Fanuc TP program (LS listing): surfaceorigin.ls

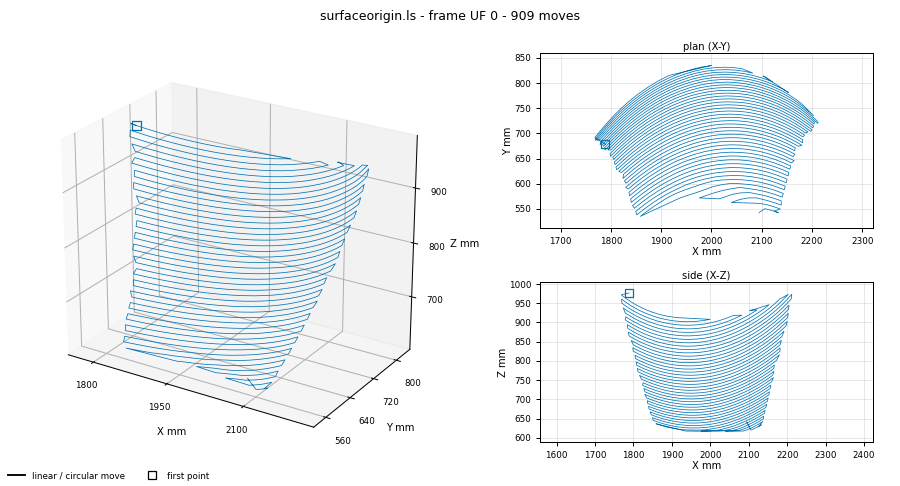
[picture p0: tool path of surfaceorigin.ls in frame UF 0, 909 of 909 moves have a stored position in this frame; points joined in program order, loops and branches not executed]
/PROG surfaceorigin
/ATTR
OWNER			= MNEDITOR;
COMMENT			= "";
PROG_SIZE		= 4757;
FILE_NAME		= surface;
VERSION			= 0;
LINE_COUNT		= 909;
MEMORY_SIZE		= 5089;
PROTECT			= READ_WRITE;
TCD:  STACK_SIZE		= 0,
      TASK_PRIORITY		= 50,
      TIME_SLICE		= 0,
      BUSY_LAMP_OFF		= 0,
      ABORT_REQUEST		= 0,
      PAUSE_REQUEST		= 0;
DEFAULT_GROUP	= 1,*,*,*,*;
CONTROL_CODE	= 00000000 00000000;
/MN
	1:  UFRAME_NUM=0 ;
	2:  UTOOL_NUM=1 ;
	3:	;
	4:	;
	5:J P[1] 100% CNT60 	;
	6:L P[2] 200mm/sec CNT60 	;
	7:L P[3] 200mm/sec CNT60 	;
	8:L P[4] 200mm/sec CNT60 	;
	9:L P[5] 200mm/sec CNT60 	;
	10:L P[6] 200mm/sec CNT60 	;
	11:L P[7] 200mm/sec CNT60 	;
	12:L P[8] 200mm/sec CNT60 	;
	13:L P[9] 200mm/sec CNT60 	;
	14:L P[10] 200mm/sec CNT60 	;
	15:L P[11] 200mm/sec CNT60 	;
	16:L P[12] 200mm/sec CNT60 	;
	17:L P[13] 200mm/sec CNT60 	;
	18:L P[14] 200mm/sec CNT60 	;
	19:L P[15] 200mm/sec CNT60 	;
	20:L P[16] 200mm/sec CNT60 	;
	21:L P[17] 200mm/sec CNT60 	;
	22:L P[18] 200mm/sec CNT60 	;
	23:L P[19] 200mm/sec CNT60 	;
	24:L P[20] 200mm/sec CNT60 	;
	25:L P[21] 200mm/sec CNT60 	;
	26:L P[22] 200mm/sec CNT60 	;
	27:L P[23] 200mm/sec CNT60 	;
	28:L P[24] 200mm/sec CNT60 	;
	29:L P[25] 200mm/sec CNT60 	;
	30:L P[26] 200mm/sec CNT60 	;
	31:L P[27] 200mm/sec CNT60 	;
	32:L P[28] 200mm/sec CNT60 	;
	33:L P[29] 200mm/sec CNT60 	;
	34:L P[30] 200mm/sec CNT60 	;
	35:L P[31] 200mm/sec CNT60 	;
	36:L P[32] 200mm/sec CNT60 	;
	37:L P[33] 200mm/sec CNT60 	;
	38:L P[34] 200mm/sec CNT60 	;
	39:L P[35] 200mm/sec CNT60 	;
	40:L P[36] 200mm/sec CNT60 	;
	41:L P[37] 200mm/sec CNT60 	;
	42:L P[38] 200mm/sec CNT60 	;
	43:L P[39] 200mm/sec CNT60 	;
	44:L P[40] 200mm/sec CNT60 	;
	45:L P[41] 200mm/sec CNT60 	;
	46:L P[42] 200mm/sec CNT60 	;
	47:L P[43] 200mm/sec CNT60 	;
	48:L P[44] 200mm/sec CNT60 	;
	49:L P[45] 200mm/sec CNT60 	;
	50:L P[46] 200mm/sec CNT60 	;
	51:L P[47] 200mm/sec CNT60 	;
	52:L P[48] 200mm/sec CNT60 	;
	53:L P[49] 200mm/sec CNT60 	;
	54:L P[50] 200mm/sec CNT60 	;
	55:L P[51] 200mm/sec CNT60 	;
	56:L P[52] 200mm/sec CNT60 	;
	57:L P[53] 200mm/sec CNT60 	;
	58:L P[54] 200mm/sec CNT60 	;
	59:L P[55] 200mm/sec CNT60 	;
	60:L P[56] 200mm/sec CNT60 	;
	61:L P[57] 200mm/sec CNT60 	;
	62:L P[58] 200mm/sec CNT60 	;
	63:L P[59] 200mm/sec CNT60 	;
	64:L P[60] 200mm/sec CNT60 	;
	65:L P[61] 200mm/sec CNT60 	;
	66:L P[62] 200mm/sec CNT60 	;
	67:L P[63] 200mm/sec CNT60 	;
	68:L P[64] 200mm/sec CNT60 	;
	69:L P[65] 200mm/sec CNT60 	;
	70:L P[66] 200mm/sec CNT60 	;
	71:L P[67] 200mm/sec CNT60 	;
	72:L P[68] 200mm/sec CNT60 	;
	73:L P[69] 200mm/sec CNT60 	;
	74:L P[70] 200mm/sec CNT60 	;
	75:L P[71] 200mm/sec CNT60 	;
	76:L P[72] 200mm/sec CNT60 	;
	77:L P[73] 200mm/sec CNT60 	;
	78:L P[74] 200mm/sec CNT60 	;
	79:L P[75] 200mm/sec CNT60 	;
	80:L P[76] 200mm/sec CNT60 	;
	81:L P[77] 200mm/sec CNT60 	;
	82:L P[78] 200mm/sec CNT60 	;
	83:L P[79] 200mm/sec CNT60 	;
	84:L P[80] 200mm/sec CNT60 	;
	85:L P[81] 200mm/sec CNT60 	;
	86:L P[82] 200mm/sec CNT60 	;
	87:L P[83] 200mm/sec CNT60 	;
	88:L P[84] 200mm/sec CNT60 	;
	89:L P[85] 200mm/sec CNT60 	;
	90:L P[86] 200mm/sec CNT60 	;
	91:L P[87] 200mm/sec CNT60 	;
	92:L P[88] 200mm/sec CNT60 	;
	93:L P[89] 200mm/sec CNT60 	;
	94:L P[90] 200mm/sec CNT60 	;
	95:L P[91] 200mm/sec CNT60 	;
	96:L P[92] 200mm/sec CNT60 	;
	97:L P[93] 200mm/sec CNT60 	;
	98:L P[94] 200mm/sec CNT60 	;
	99:L P[95] 200mm/sec CNT60 	;
	100:L P[96] 200mm/sec CNT60 	;
	101:L P[97] 200mm/sec CNT60 	;
	102:L P[98] 200mm/sec CNT60 	;
	103:L P[99] 200mm/sec CNT60 	;
	104:L P[100] 200mm/sec CNT60 	;
	105:L P[101] 200mm/sec CNT60 	;
	106:L P[102] 200mm/sec CNT60 	;
	107:L P[103] 200mm/sec CNT60 	;
	108:L P[104] 200mm/sec CNT60 	;
	109:L P[105] 200mm/sec CNT60 	;
	110:L P[106] 200mm/sec CNT60 	;
	111:L P[107] 200mm/sec CNT60 	;
	112:L P[108] 200mm/sec CNT60 	;
	113:L P[109] 200mm/sec CNT60 	;
	114:L P[110] 200mm/sec CNT60 	;
	115:L P[111] 200mm/sec CNT60 	;
	116:L P[112] 200mm/sec CNT60 	;
	117:L P[113] 200mm/sec CNT60 	;
	118:L P[114] 200mm/sec CNT60 	;
	119:L P[115] 200mm/sec CNT60 	;
	120:L P[116] 200mm/sec CNT60 	;
	121:L P[117] 200mm/sec CNT60 	;
	122:L P[118] 200mm/sec CNT60 	;
	123:L P[119] 200mm/sec CNT60 	;
	124:L P[120] 200mm/sec CNT60 	;
	125:L P[121] 200mm/sec CNT60 	;
	126:L P[122] 200mm/sec CNT60 	;
	127:L P[123] 200mm/sec CNT60 	;
	128:L P[124] 200mm/sec CNT60 	;
	129:L P[125] 200mm/sec CNT60 	;
	130:L P[126] 200mm/sec CNT60 	;
	131:L P[127] 200mm/sec CNT60 	;
	132:L P[128] 200mm/sec CNT60 	;
	133:L P[129] 200mm/sec CNT60 	;
	134:L P[130] 200mm/sec CNT60 	;
	135:L P[131] 200mm/sec CNT60 	;
	136:L P[132] 200mm/sec CNT60 	;
	137:L P[133] 200mm/sec CNT60 	;
	138:L P[134] 200mm/sec CNT60 	;
	139:L P[135] 200mm/sec CNT60 	;
	140:L P[136] 200mm/sec CNT60 	;
	141:L P[137] 200mm/sec CNT60 	;
	142:L P[138] 200mm/sec CNT60 	;
	143:L P[139] 200mm/sec CNT60 	;
	144:L P[140] 200mm/sec CNT60 	;
	145:L P[141] 200mm/sec CNT60 	;
	146:L P[142] 200mm/sec CNT60 	;
	147:L P[143] 200mm/sec CNT60 	;
	148:L P[144] 200mm/sec CNT60 	;
	149:L P[145] 200mm/sec CNT60 	;
	150:L P[146] 200mm/sec CNT60 	;
	151:L P[147] 200mm/sec CNT60 	;
	152:L P[148] 200mm/sec CNT60 	;
	153:L P[149] 200mm/sec CNT60 	;
	154:L P[150] 200mm/sec CNT60 	;
	155:L P[151] 200mm/sec CNT60 	;
	156:L P[152] 200mm/sec CNT60 	;
	157:L P[153] 200mm/sec CNT60 	;
	158:L P[154] 200mm/sec CNT60 	;
	159:L P[155] 200mm/sec CNT60 	;
	160:L P[156] 200mm/sec CNT60 	;
	161:L P[157] 200mm/sec CNT60 	;
	162:L P[158] 200mm/sec CNT60 	;
	163:L P[159] 200mm/sec CNT60 	;
	164:L P[160] 200mm/sec CNT60 	;
	165:L P[161] 200mm/sec CNT60 	;
	166:L P[162] 200mm/sec CNT60 	;
	167:L P[163] 200mm/sec CNT60 	;
	168:L P[164] 200mm/sec CNT60 	;
	169:L P[165] 200mm/sec CNT60 	;
	170:L P[166] 200mm/sec CNT60 	;
	171:L P[167] 200mm/sec CNT60 	;
	172:L P[168] 200mm/sec CNT60 	;
	173:L P[169] 200mm/sec CNT60 	;
	174:L P[170] 200mm/sec CNT60 	;
	175:L P[171] 200mm/sec CNT60 	;
	176:L P[172] 200mm/sec CNT60 	;
	177:L P[173] 200mm/sec CNT60 	;
	178:L P[174] 200mm/sec CNT60 	;
	179:L P[175] 200mm/sec CNT60 	;
	180:L P[176] 200mm/sec CNT60 	;
	181:L P[177] 200mm/sec CNT60 	;
	182:L P[178] 200mm/sec CNT60 	;
	183:L P[179] 200mm/sec CNT60 	;
	184:L P[180] 200mm/sec CNT60 	;
	185:L P[181] 200mm/sec CNT60 	;
	186:L P[182] 200mm/sec CNT60 	;
	187:L P[183] 200mm/sec CNT60 	;
	188:L P[184] 200mm/sec CNT60 	;
	189:L P[185] 200mm/sec CNT60 	;
	190:L P[186] 200mm/sec CNT60 	;
	191:L P[187] 200mm/sec CNT60 	;
	192:L P[188] 200mm/sec CNT60 	;
	193:L P[189] 200mm/sec CNT60 	;
	194:L P[190] 200mm/sec CNT60 	;
	195:L P[191] 200mm/sec CNT60 	;
	196:L P[192] 200mm/sec CNT60 	;
	197:L P[193] 200mm/sec CNT60 	;
	198:L P[194] 200mm/sec CNT60 	;
	199:L P[195] 200mm/sec CNT60 	;
	200:L P[196] 200mm/sec CNT60 	;
	201:L P[197] 200mm/sec CNT60 	;
	202:L P[198] 200mm/sec CNT60 	;
	203:L P[199] 200mm/sec CNT60 	;
	204:L P[200] 200mm/sec CNT60 	;
	205:L P[201] 200mm/sec CNT60 	;
	206:L P[202] 200mm/sec CNT60 	;
	207:L P[203] 200mm/sec CNT60 	;
	208:L P[204] 200mm/sec CNT60 	;
	209:L P[205] 200mm/sec CNT60 	;
	210:L P[206] 200mm/sec CNT60 	;
	211:L P[207] 200mm/sec CNT60 	;
	212:L P[208] 200mm/sec CNT60 	;
	213:L P[209] 200mm/sec CNT60 	;
	214:L P[210] 200mm/sec CNT60 	;
	215:L P[211] 200mm/sec CNT60 	;
	216:L P[212] 200mm/sec CNT60 	;
	217:L P[213] 200mm/sec CNT60 	;
	218:L P[214] 200mm/sec CNT60 	;
	219:L P[215] 200mm/sec CNT60 	;
	220:L P[216] 200mm/sec CNT60 	;
	221:L P[217] 200mm/sec CNT60 	;
	222:L P[218] 200mm/sec CNT60 	;
	223:L P[219] 200mm/sec CNT60 	;
	224:L P[220] 200mm/sec CNT60 	;
	225:L P[221] 200mm/sec CNT60 	;
	226:L P[222] 200mm/sec CNT60 	;
	227:L P[223] 200mm/sec CNT60 	;
	228:L P[224] 200mm/sec CNT60 	;
	229:L P[225] 200mm/sec CNT60 	;
	230:L P[226] 200mm/sec CNT60 	;
	231:L P[227] 200mm/sec CNT60 	;
	232:L P[228] 200mm/sec CNT60 	;
	233:L P[229] 200mm/sec CNT60 	;
	234:L P[230] 200mm/sec CNT60 	;
	235:L P[231] 200mm/sec CNT60 	;
	236:L P[232] 200mm/sec CNT60 	;
	237:L P[233] 200mm/sec CNT60 	;
	238:L P[234] 200mm/sec CNT60 	;
	239:L P[235] 200mm/sec CNT60 	;
	240:L P[236] 200mm/sec CNT60 	;
	241:L P[237] 200mm/sec CNT60 	;
	242:L P[238] 200mm/sec CNT60 	;
	243:L P[239] 200mm/sec CNT60 	;
	244:L P[240] 200mm/sec CNT60 	;
	245:L P[241] 200mm/sec CNT60 	;
	246:L P[242] 200mm/sec CNT60 	;
	247:L P[243] 200mm/sec CNT60 	;
	248:L P[244] 200mm/sec CNT60 	;
	249:L P[245] 200mm/sec CNT60 	;
	250:L P[246] 200mm/sec CNT60 	;
	251:L P[247] 200mm/sec CNT60 	;
	252:L P[248] 200mm/sec CNT60 	;
	253:L P[249] 200mm/sec CNT60 	;
	254:L P[250] 200mm/sec CNT60 	;
	255:L P[251] 200mm/sec CNT60 	;
	256:L P[252] 200mm/sec CNT60 	;
	257:L P[253] 200mm/sec CNT60 	;
	258:L P[254] 200mm/sec CNT60 	;
	259:L P[255] 200mm/sec CNT60 	;
	260:L P[256] 200mm/sec CNT60 	;
	261:L P[257] 200mm/sec CNT60 	;
	262:L P[258] 200mm/sec CNT60 	;
	263:L P[259] 200mm/sec CNT60 	;
	264:L P[260] 200mm/sec CNT60 	;
	265:L P[261] 200mm/sec CNT60 	;
	266:L P[262] 200mm/sec CNT60 	;
	267:L P[263] 200mm/sec CNT60 	;
	268:L P[264] 200mm/sec CNT60 	;
	269:L P[265] 200mm/sec CNT60 	;
	270:L P[266] 200mm/sec CNT60 	;
	271:L P[267] 200mm/sec CNT60 	;
	272:L P[268] 200mm/sec CNT60 	;
	273:L P[269] 200mm/sec CNT60 	;
	274:L P[270] 200mm/sec CNT60 	;
	275:L P[271] 200mm/sec CNT60 	;
	276:L P[272] 200mm/sec CNT60 	;
	277:L P[273] 200mm/sec CNT60 	;
	278:L P[274] 200mm/sec CNT60 	;
	279:L P[275] 200mm/sec CNT60 	;
	280:L P[276] 200mm/sec CNT60 	;
	281:L P[277] 200mm/sec CNT60 	;
	282:L P[278] 200mm/sec CNT60 	;
	283:L P[279] 200mm/sec CNT60 	;
	284:L P[280] 200mm/sec CNT60 	;
	285:L P[281] 200mm/sec CNT60 	;
	286:L P[282] 200mm/sec CNT60 	;
	287:L P[283] 200mm/sec CNT60 	;
	288:L P[284] 200mm/sec CNT60 	;
	289:L P[285] 200mm/sec CNT60 	;
	290:L P[286] 200mm/sec CNT60 	;
	291:L P[287] 200mm/sec CNT60 	;
	292:L P[288] 200mm/sec CNT60 	;
	293:L P[289] 200mm/sec CNT60 	;
	294:L P[290] 200mm/sec CNT60 	;
	295:L P[291] 200mm/sec CNT60 	;
	296:L P[292] 200mm/sec CNT60 	;
	297:L P[293] 200mm/sec CNT60 	;
	298:L P[294] 200mm/sec CNT60 	;
	299:L P[295] 200mm/sec CNT60 	;
	300:L P[296] 200mm/sec CNT60 	;
	301:L P[297] 200mm/sec CNT60 	;
	302:L P[298] 200mm/sec CNT60 	;
	303:L P[299] 200mm/sec CNT60 	;
	304:L P[300] 200mm/sec CNT60 	;
	305:L P[301] 200mm/sec CNT60 	;
	306:L P[302] 200mm/sec CNT60 	;
	307:L P[303] 200mm/sec CNT60 	;
	308:L P[304] 200mm/sec CNT60 	;
	309:L P[305] 200mm/sec CNT60 	;
	310:L P[306] 200mm/sec CNT60 	;
	311:L P[307] 200mm/sec CNT60 	;
	312:L P[308] 200mm/sec CNT60 	;
	313:L P[309] 200mm/sec CNT60 	;
	314:L P[310] 200mm/sec CNT60 	;
	315:L P[311] 200mm/sec CNT60 	;
	316:L P[312] 200mm/sec CNT60 	;
	317:L P[313] 200mm/sec CNT60 	;
	318:L P[314] 200mm/sec CNT60 	;
	319:L P[315] 200mm/sec CNT60 	;
	320:L P[316] 200mm/sec CNT60 	;
	321:L P[317] 200mm/sec CNT60 	;
	322:L P[318] 200mm/sec CNT60 	;
	323:L P[319] 200mm/sec CNT60 	;
	324:L P[320] 200mm/sec CNT60 	;
	325:L P[321] 200mm/sec CNT60 	;
	326:L P[322] 200mm/sec CNT60 	;
	327:L P[323] 200mm/sec CNT60 	;
	328:L P[324] 200mm/sec CNT60 	;
	329:L P[325] 200mm/sec CNT60 	;
	330:L P[326] 200mm/sec CNT60 	;
	331:L P[327] 200mm/sec CNT60 	;
	332:L P[328] 200mm/sec CNT60 	;
	333:L P[329] 200mm/sec CNT60 	;
	334:L P[330] 200mm/sec CNT60 	;
	335:L P[331] 200mm/sec CNT60 	;
	336:L P[332] 200mm/sec CNT60 	;
	337:L P[333] 200mm/sec CNT60 	;
	338:L P[334] 200mm/sec CNT60 	;
	339:L P[335] 200mm/sec CNT60 	;
	340:L P[336] 200mm/sec CNT60 	;
	341:L P[337] 200mm/sec CNT60 	;
	342:L P[338] 200mm/sec CNT60 	;
	343:L P[339] 200mm/sec CNT60 	;
	344:L P[340] 200mm/sec CNT60 	;
	345:L P[341] 200mm/sec CNT60 	;
	346:L P[342] 200mm/sec CNT60 	;
	347:L P[343] 200mm/sec CNT60 	;
	348:L P[344] 200mm/sec CNT60 	;
	349:L P[345] 200mm/sec CNT60 	;
	350:L P[346] 200mm/sec CNT60 	;
	351:L P[347] 200mm/sec CNT60 	;
	352:L P[348] 200mm/sec CNT60 	;
	353:L P[349] 200mm/sec CNT60 	;
	354:L P[350] 200mm/sec CNT60 	;
	355:L P[351] 200mm/sec CNT60 	;
	356:L P[352] 200mm/sec CNT60 	;
	357:L P[353] 200mm/sec CNT60 	;
	358:L P[354] 200mm/sec CNT60 	;
	359:L P[355] 200mm/sec CNT60 	;
	360:L P[356] 200mm/sec CNT60 	;
	361:L P[357] 200mm/sec CNT60 	;
	362:L P[358] 200mm/sec CNT60 	;
	363:L P[359] 200mm/sec CNT60 	;
	364:L P[360] 200mm/sec CNT60 	;
	365:L P[361] 200mm/sec CNT60 	;
	366:L P[362] 200mm/sec CNT60 	;
	367:L P[363] 200mm/sec CNT60 	;
	368:L P[364] 200mm/sec CNT60 	;
	369:L P[365] 200mm/sec CNT60 	;
	370:L P[366] 200mm/sec CNT60 	;
	371:L P[367] 200mm/sec CNT60 	;
	372:L P[368] 200mm/sec CNT60 	;
	373:L P[369] 200mm/sec CNT60 	;
	374:L P[370] 200mm/sec CNT60 	;
	375:L P[371] 200mm/sec CNT60 	;
	376:L P[372] 200mm/sec CNT60 	;
	377:L P[373] 200mm/sec CNT60 	;
	378:L P[374] 200mm/sec CNT60 	;
	379:L P[375] 200mm/sec CNT60 	;
	380:L P[376] 200mm/sec CNT60 	;
	381:L P[377] 200mm/sec CNT60 	;
	382:L P[378] 200mm/sec CNT60 	;
	383:L P[379] 200mm/sec CNT60 	;
	384:L P[380] 200mm/sec CNT60 	;
	385:L P[381] 200mm/sec CNT60 	;
	386:L P[382] 200mm/sec CNT60 	;
	387:L P[383] 200mm/sec CNT60 	;
	388:L P[384] 200mm/sec CNT60 	;
	389:L P[385] 200mm/sec CNT60 	;
	390:L P[386] 200mm/sec CNT60 	;
	391:L P[387] 200mm/sec CNT60 	;
	392:L P[388] 200mm/sec CNT60 	;
	393:L P[389] 200mm/sec CNT60 	;
	394:L P[390] 200mm/sec CNT60 	;
	395:L P[391] 200mm/sec CNT60 	;
	396:L P[392] 200mm/sec CNT60 	;
	397:L P[393] 200mm/sec CNT60 	;
	398:L P[394] 200mm/sec CNT60 	;
	399:L P[395] 200mm/sec CNT60 	;
	400:L P[396] 200mm/sec CNT60 	;
	401:L P[397] 200mm/sec CNT60 	;
	402:L P[398] 200mm/sec CNT60 	;
	403:L P[399] 200mm/sec CNT60 	;
	404:L P[400] 200mm/sec CNT60 	;
	405:L P[401] 200mm/sec CNT60 	;
	406:L P[402] 200mm/sec CNT60 	;
	407:L P[403] 200mm/sec CNT60 	;
	408:L P[404] 200mm/sec CNT60 	;
	409:L P[405] 200mm/sec CNT60 	;
	410:L P[406] 200mm/sec CNT60 	;
	411:L P[407] 200mm/sec CNT60 	;
	412:L P[408] 200mm/sec CNT60 	;
	413:L P[409] 200mm/sec CNT60 	;
	414:L P[410] 200mm/sec CNT60 	;
	415:L P[411] 200mm/sec CNT60 	;
	416:L P[412] 200mm/sec CNT60 	;
	417:L P[413] 200mm/sec CNT60 	;
	418:L P[414] 200mm/sec CNT60 	;
	419:L P[415] 200mm/sec CNT60 	;
	420:L P[416] 200mm/sec CNT60 	;
	421:L P[417] 200mm/sec CNT60 	;
	422:L P[418] 200mm/sec CNT60 	;
	423:L P[419] 200mm/sec CNT60 	;
	424:L P[420] 200mm/sec CNT60 	;
	425:L P[421] 200mm/sec CNT60 	;
	426:L P[422] 200mm/sec CNT60 	;
	427:L P[423] 200mm/sec CNT60 	;
	428:L P[424] 200mm/sec CNT60 	;
	429:L P[425] 200mm/sec CNT60 	;
	430:L P[426] 200mm/sec CNT60 	;
	431:L P[427] 200mm/sec CNT60 	;
	432:L P[428] 200mm/sec CNT60 	;
	433:L P[429] 200mm/sec CNT60 	;
	434:L P[430] 200mm/sec CNT60 	;
	435:L P[431] 200mm/sec CNT60 	;
	436:L P[432] 200mm/sec CNT60 	;
	437:L P[433] 200mm/sec CNT60 	;
	438:L P[434] 200mm/sec CNT60 	;
	439:L P[435] 200mm/sec CNT60 	;
	440:L P[436] 200mm/sec CNT60 	;
	441:L P[437] 200mm/sec CNT60 	;
	442:L P[438] 200mm/sec CNT60 	;
	443:L P[439] 200mm/sec CNT60 	;
	444:L P[440] 200mm/sec CNT60 	;
	445:L P[441] 200mm/sec CNT60 	;
	446:L P[442] 200mm/sec CNT60 	;
	447:L P[443] 200mm/sec CNT60 	;
	448:L P[444] 200mm/sec CNT60 	;
	449:L P[445] 200mm/sec CNT60 	;
	450:L P[446] 200mm/sec CNT60 	;
	451:L P[447] 200mm/sec CNT60 	;
	452:L P[448] 200mm/sec CNT60 	;
	453:L P[449] 200mm/sec CNT60 	;
	454:L P[450] 200mm/sec CNT60 	;
	455:L P[451] 200mm/sec CNT60 	;
	456:L P[452] 200mm/sec CNT60 	;
	457:L P[453] 200mm/sec CNT60 	;
	458:L P[454] 200mm/sec CNT60 	;
	459:L P[455] 200mm/sec CNT60 	;
	460:L P[456] 200mm/sec CNT60 	;
	461:L P[457] 200mm/sec CNT60 	;
	462:L P[458] 200mm/sec CNT60 	;
	463:L P[459] 200mm/sec CNT60 	;
	464:L P[460] 200mm/sec CNT60 	;
	465:L P[461] 200mm/sec CNT60 	;
	466:L P[462] 200mm/sec CNT60 	;
	467:L P[463] 200mm/sec CNT60 	;
	468:L P[464] 200mm/sec CNT60 	;
	469:L P[465] 200mm/sec CNT60 	;
	470:L P[466] 200mm/sec CNT60 	;
	471:L P[467] 200mm/sec CNT60 	;
	472:L P[468] 200mm/sec CNT60 	;
	473:L P[469] 200mm/sec CNT60 	;
	474:L P[470] 200mm/sec CNT60 	;
	475:L P[471] 200mm/sec CNT60 	;
	476:L P[472] 200mm/sec CNT60 	;
	477:L P[473] 200mm/sec CNT60 	;
	478:L P[474] 200mm/sec CNT60 	;
	479:L P[475] 200mm/sec CNT60 	;
	480:L P[476] 200mm/sec CNT60 	;
	481:L P[477] 200mm/sec CNT60 	;
	482:L P[478] 200mm/sec CNT60 	;
	483:L P[479] 200mm/sec CNT60 	;
	484:L P[480] 200mm/sec CNT60 	;
	485:L P[481] 200mm/sec CNT60 	;
	486:L P[482] 200mm/sec CNT60 	;
	487:L P[483] 200mm/sec CNT60 	;
	488:L P[484] 200mm/sec CNT60 	;
	489:L P[485] 200mm/sec CNT60 	;
	490:L P[486] 200mm/sec CNT60 	;
	491:L P[487] 200mm/sec CNT60 	;
	492:L P[488] 200mm/sec CNT60 	;
	493:L P[489] 200mm/sec CNT60 	;
	494:L P[490] 200mm/sec CNT60 	;
	495:L P[491] 200mm/sec CNT60 	;
	496:L P[492] 200mm/sec CNT60 	;
	497:L P[493] 200mm/sec CNT60 	;
	498:L P[494] 200mm/sec CNT60 	;
	499:L P[495] 200mm/sec CNT60 	;
	500:L P[496] 200mm/sec CNT60 	;
	501:L P[497] 200mm/sec CNT60 	;
	502:L P[498] 200mm/sec CNT60 	;
	503:L P[499] 200mm/sec CNT60 	;
	504:L P[500] 200mm/sec CNT60 	;
	505:L P[501] 200mm/sec CNT60 	;
	506:L P[502] 200mm/sec CNT60 	;
	507:L P[503] 200mm/sec CNT60 	;
	508:L P[504] 200mm/sec CNT60 	;
	509:L P[505] 200mm/sec CNT60 	;
	510:L P[506] 200mm/sec CNT60 	;
	511:L P[507] 200mm/sec CNT60 	;
	512:L P[508] 200mm/sec CNT60 	;
	513:L P[509] 200mm/sec CNT60 	;
	514:L P[510] 200mm/sec CNT60 	;
	515:L P[511] 200mm/sec CNT60 	;
	516:L P[512] 200mm/sec CNT60 	;
	517:L P[513] 200mm/sec CNT60 	;
	518:L P[514] 200mm/sec CNT60 	;
	519:L P[515] 200mm/sec CNT60 	;
	520:L P[516] 200mm/sec CNT60 	;
	521:L P[517] 200mm/sec CNT60 	;
	522:L P[518] 200mm/sec CNT60 	;
	523:L P[519] 200mm/sec CNT60 	;
	524:L P[520] 200mm/sec CNT60 	;
	525:L P[521] 200mm/sec CNT60 	;
	526:L P[522] 200mm/sec CNT60 	;
	527:L P[523] 200mm/sec CNT60 	;
	528:L P[524] 200mm/sec CNT60 	;
	529:L P[525] 200mm/sec CNT60 	;
	530:L P[526] 200mm/sec CNT60 	;
	531:L P[527] 200mm/sec CNT60 	;
	532:L P[528] 200mm/sec CNT60 	;
	533:L P[529] 200mm/sec CNT60 	;
	534:L P[530] 200mm/sec CNT60 	;
	535:L P[531] 200mm/sec CNT60 	;
	536:L P[532] 200mm/sec CNT60 	;
	537:L P[533] 200mm/sec CNT60 	;
	538:L P[534] 200mm/sec CNT60 	;
	539:L P[535] 200mm/sec CNT60 	;
	540:L P[536] 200mm/sec CNT60 	;
	541:L P[537] 200mm/sec CNT60 	;
	542:L P[538] 200mm/sec CNT60 	;
	543:L P[539] 200mm/sec CNT60 	;
	544:L P[540] 200mm/sec CNT60 	;
	545:L P[541] 200mm/sec CNT60 	;
	546:L P[542] 200mm/sec CNT60 	;
	547:L P[543] 200mm/sec CNT60 	;
	548:L P[544] 200mm/sec CNT60 	;
	549:L P[545] 200mm/sec CNT60 	;
	550:L P[546] 200mm/sec CNT60 	;
	551:L P[547] 200mm/sec CNT60 	;
	552:L P[548] 200mm/sec CNT60 	;
	553:L P[549] 200mm/sec CNT60 	;
	554:L P[550] 200mm/sec CNT60 	;
	555:L P[551] 200mm/sec CNT60 	;
	556:L P[552] 200mm/sec CNT60 	;
	557:L P[553] 200mm/sec CNT60 	;
	558:L P[554] 200mm/sec CNT60 	;
	559:L P[555] 200mm/sec CNT60 	;
	560:L P[556] 200mm/sec CNT60 	;
	561:L P[557] 200mm/sec CNT60 	;
	562:L P[558] 200mm/sec CNT60 	;
	563:L P[559] 200mm/sec CNT60 	;
	564:L P[560] 200mm/sec CNT60 	;
	565:L P[561] 200mm/sec CNT60 	;
	566:L P[562] 200mm/sec CNT60 	;
	567:L P[563] 200mm/sec CNT60 	;
	568:L P[564] 200mm/sec CNT60 	;
	569:L P[565] 200mm/sec CNT60 	;
	570:L P[566] 200mm/sec CNT60 	;
	571:L P[567] 200mm/sec CNT60 	;
	572:L P[568] 200mm/sec CNT60 	;
	573:L P[569] 200mm/sec CNT60 	;
	574:L P[570] 200mm/sec CNT60 	;
	575:L P[571] 200mm/sec CNT60 	;
	576:L P[572] 200mm/sec CNT60 	;
	577:L P[573] 200mm/sec CNT60 	;
	578:L P[574] 200mm/sec CNT60 	;
	579:L P[575] 200mm/sec CNT60 	;
	580:L P[576] 200mm/sec CNT60 	;
	581:L P[577] 200mm/sec CNT60 	;
	582:L P[578] 200mm/sec CNT60 	;
	583:L P[579] 200mm/sec CNT60 	;
	584:L P[580] 200mm/sec CNT60 	;
	585:L P[581] 200mm/sec CNT60 	;
	586:L P[582] 200mm/sec CNT60 	;
	587:L P[583] 200mm/sec CNT60 	;
	588:L P[584] 200mm/sec CNT60 	;
	589:L P[585] 200mm/sec CNT60 	;
	590:L P[586] 200mm/sec CNT60 	;
	591:L P[587] 200mm/sec CNT60 	;
	592:L P[588] 200mm/sec CNT60 	;
	593:L P[589] 200mm/sec CNT60 	;
	594:L P[590] 200mm/sec CNT60 	;
	595:L P[591] 200mm/sec CNT60 	;
	596:L P[592] 200mm/sec CNT60 	;
	597:L P[593] 200mm/sec CNT60 	;
	598:L P[594] 200mm/sec CNT60 	;
	599:L P[595] 200mm/sec CNT60 	;
	600:L P[596] 200mm/sec CNT60 	;
	601:L P[597] 200mm/sec CNT60 	;
	602:L P[598] 200mm/sec CNT60 	;
	603:L P[599] 200mm/sec CNT60 	;
	604:L P[600] 200mm/sec CNT60 	;
	605:L P[601] 200mm/sec CNT60 	;
	606:L P[602] 200mm/sec CNT60 	;
	607:L P[603] 200mm/sec CNT60 	;
	608:L P[604] 200mm/sec CNT60 	;
	609:L P[605] 200mm/sec CNT60 	;
	610:L P[606] 200mm/sec CNT60 	;
	611:L P[607] 200mm/sec CNT60 	;
	612:L P[608] 200mm/sec CNT60 	;
	613:L P[609] 200mm/sec CNT60 	;
	614:L P[610] 200mm/sec CNT60 	;
	615:L P[611] 200mm/sec CNT60 	;
	616:L P[612] 200mm/sec CNT60 	;
	617:L P[613] 200mm/sec CNT60 	;
	618:L P[614] 200mm/sec CNT60 	;
	619:L P[615] 200mm/sec CNT60 	;
	620:L P[616] 200mm/sec CNT60 	;
	621:L P[617] 200mm/sec CNT60 	;
	622:L P[618] 200mm/sec CNT60 	;
	623:L P[619] 200mm/sec CNT60 	;
	624:L P[620] 200mm/sec CNT60 	;
	625:L P[621] 200mm/sec CNT60 	;
	626:L P[622] 200mm/sec CNT60 	;
	627:L P[623] 200mm/sec CNT60 	;
	628:L P[624] 200mm/sec CNT60 	;
	629:L P[625] 200mm/sec CNT60 	;
	630:L P[626] 200mm/sec CNT60 	;
	631:L P[627] 200mm/sec CNT60 	;
	632:L P[628] 200mm/sec CNT60 	;
	633:L P[629] 200mm/sec CNT60 	;
	634:L P[630] 200mm/sec CNT60 	;
	635:L P[631] 200mm/sec CNT60 	;
	636:L P[632] 200mm/sec CNT60 	;
	637:L P[633] 200mm/sec CNT60 	;
	638:L P[634] 200mm/sec CNT60 	;
	639:L P[635] 200mm/sec CNT60 	;
	640:L P[636] 200mm/sec CNT60 	;
	641:L P[637] 200mm/sec CNT60 	;
	642:L P[638] 200mm/sec CNT60 	;
	643:L P[639] 200mm/sec CNT60 	;
	644:L P[640] 200mm/sec CNT60 	;
	645:L P[641] 200mm/sec CNT60 	;
	646:L P[642] 200mm/sec CNT60 	;
	647:L P[643] 200mm/sec CNT60 	;
	648:L P[644] 200mm/sec CNT60 	;
	649:L P[645] 200mm/sec CNT60 	;
	650:L P[646] 200mm/sec CNT60 	;
	651:L P[647] 200mm/sec CNT60 	;
	652:L P[648] 200mm/sec CNT60 	;
	653:L P[649] 200mm/sec CNT60 	;
	654:L P[650] 200mm/sec CNT60 	;
	655:L P[651] 200mm/sec CNT60 	;
	656:L P[652] 200mm/sec CNT60 	;
	657:L P[653] 200mm/sec CNT60 	;
	658:L P[654] 200mm/sec CNT60 	;
	659:L P[655] 200mm/sec CNT60 	;
	660:L P[656] 200mm/sec CNT60 	;
	661:L P[657] 200mm/sec CNT60 	;
	662:L P[658] 200mm/sec CNT60 	;
	663:L P[659] 200mm/sec CNT60 	;
	664:L P[660] 200mm/sec CNT60 	;
	665:L P[661] 200mm/sec CNT60 	;
	666:L P[662] 200mm/sec CNT60 	;
	667:L P[663] 200mm/sec CNT60 	;
	668:L P[664] 200mm/sec CNT60 	;
	669:L P[665] 200mm/sec CNT60 	;
	670:L P[666] 200mm/sec CNT60 	;
	671:L P[667] 200mm/sec CNT60 	;
	672:L P[668] 200mm/sec CNT60 	;
	673:L P[669] 200mm/sec CNT60 	;
	674:L P[670] 200mm/sec CNT60 	;
	675:L P[671] 200mm/sec CNT60 	;
	676:L P[672] 200mm/sec CNT60 	;
	677:L P[673] 200mm/sec CNT60 	;
	678:L P[674] 200mm/sec CNT60 	;
	679:L P[675] 200mm/sec CNT60 	;
	680:L P[676] 200mm/sec CNT60 	;
	681:L P[677] 200mm/sec CNT60 	;
	682:L P[678] 200mm/sec CNT60 	;
	683:L P[679] 200mm/sec CNT60 	;
	684:L P[680] 200mm/sec CNT60 	;
	685:L P[681] 200mm/sec CNT60 	;
	686:L P[682] 200mm/sec CNT60 	;
	687:L P[683] 200mm/sec CNT60 	;
	688:L P[684] 200mm/sec CNT60 	;
	689:L P[685] 200mm/sec CNT60 	;
	690:L P[686] 200mm/sec CNT60 	;
	691:L P[687] 200mm/sec CNT60 	;
	692:L P[688] 200mm/sec CNT60 	;
	693:L P[689] 200mm/sec CNT60 	;
	694:L P[690] 200mm/sec CNT60 	;
	695:L P[691] 200mm/sec CNT60 	;
	696:L P[692] 200mm/sec CNT60 	;
	697:L P[693] 200mm/sec CNT60 	;
	698:L P[694] 200mm/sec CNT60 	;
	699:L P[695] 200mm/sec CNT60 	;
	700:L P[696] 200mm/sec CNT60 	;
	701:L P[697] 200mm/sec CNT60 	;
	702:L P[698] 200mm/sec CNT60 	;
	703:L P[699] 200mm/sec CNT60 	;
	704:L P[700] 200mm/sec CNT60 	;
	705:L P[701] 200mm/sec CNT60 	;
	706:L P[702] 200mm/sec CNT60 	;
	707:L P[703] 200mm/sec CNT60 	;
	708:L P[704] 200mm/sec CNT60 	;
	709:L P[705] 200mm/sec CNT60 	;
	710:L P[706] 200mm/sec CNT60 	;
	711:L P[707] 200mm/sec CNT60 	;
	712:L P[708] 200mm/sec CNT60 	;
	713:L P[709] 200mm/sec CNT60 	;
	714:L P[710] 200mm/sec CNT60 	;
	715:L P[711] 200mm/sec CNT60 	;
	716:L P[712] 200mm/sec CNT60 	;
	717:L P[713] 200mm/sec CNT60 	;
	718:L P[714] 200mm/sec CNT60 	;
	719:L P[715] 200mm/sec CNT60 	;
	720:L P[716] 200mm/sec CNT60 	;
	721:L P[717] 200mm/sec CNT60 	;
	722:L P[718] 200mm/sec CNT60 	;
	723:L P[719] 200mm/sec CNT60 	;
	724:L P[720] 200mm/sec CNT60 	;
	725:L P[721] 200mm/sec CNT60 	;
	726:L P[722] 200mm/sec CNT60 	;
	727:L P[723] 200mm/sec CNT60 	;
	728:L P[724] 200mm/sec CNT60 	;
	729:L P[725] 200mm/sec CNT60 	;
	730:L P[726] 200mm/sec CNT60 	;
	731:L P[727] 200mm/sec CNT60 	;
	732:L P[728] 200mm/sec CNT60 	;
	733:L P[729] 200mm/sec CNT60 	;
	734:L P[730] 200mm/sec CNT60 	;
	735:L P[731] 200mm/sec CNT60 	;
	736:L P[732] 200mm/sec CNT60 	;
	737:L P[733] 200mm/sec CNT60 	;
	738:L P[734] 200mm/sec CNT60 	;
	739:L P[735] 200mm/sec CNT60 	;
	740:L P[736] 200mm/sec CNT60 	;
	741:L P[737] 200mm/sec CNT60 	;
	742:L P[738] 200mm/sec CNT60 	;
	743:L P[739] 200mm/sec CNT60 	;
	744:L P[740] 200mm/sec CNT60 	;
	745:L P[741] 200mm/sec CNT60 	;
	746:L P[742] 200mm/sec CNT60 	;
	747:L P[743] 200mm/sec CNT60 	;
	748:L P[744] 200mm/sec CNT60 	;
	749:L P[745] 200mm/sec CNT60 	;
	750:L P[746] 200mm/sec CNT60 	;
	751:L P[747] 200mm/sec CNT60 	;
	752:L P[748] 200mm/sec CNT60 	;
	753:L P[749] 200mm/sec CNT60 	;
	754:L P[750] 200mm/sec CNT60 	;
	755:L P[751] 200mm/sec CNT60 	;
	756:L P[752] 200mm/sec CNT60 	;
	757:L P[753] 200mm/sec CNT60 	;
	758:L P[754] 200mm/sec CNT60 	;
	759:L P[755] 200mm/sec CNT60 	;
	760:L P[756] 200mm/sec CNT60 	;
	761:L P[757] 200mm/sec CNT60 	;
	762:L P[758] 200mm/sec CNT60 	;
	763:L P[759] 200mm/sec CNT60 	;
	764:L P[760] 200mm/sec CNT60 	;
	765:L P[761] 200mm/sec CNT60 	;
	766:L P[762] 200mm/sec CNT60 	;
	767:L P[763] 200mm/sec CNT60 	;
	768:L P[764] 200mm/sec CNT60 	;
	769:L P[765] 200mm/sec CNT60 	;
	770:L P[766] 200mm/sec CNT60 	;
	771:L P[767] 200mm/sec CNT60 	;
	772:L P[768] 200mm/sec CNT60 	;
	773:L P[769] 200mm/sec CNT60 	;
	774:L P[770] 200mm/sec CNT60 	;
	775:L P[771] 200mm/sec CNT60 	;
	776:L P[772] 200mm/sec CNT60 	;
	777:L P[773] 200mm/sec CNT60 	;
	778:L P[774] 200mm/sec CNT60 	;
	779:L P[775] 200mm/sec CNT60 	;
	780:L P[776] 200mm/sec CNT60 	;
	781:L P[777] 200mm/sec CNT60 	;
	782:L P[778] 200mm/sec CNT60 	;
	783:L P[779] 200mm/sec CNT60 	;
	784:L P[780] 200mm/sec CNT60 	;
	785:L P[781] 200mm/sec CNT60 	;
	786:L P[782] 200mm/sec CNT60 	;
	787:L P[783] 200mm/sec CNT60 	;
	788:L P[784] 200mm/sec CNT60 	;
	789:L P[785] 200mm/sec CNT60 	;
	790:L P[786] 200mm/sec CNT60 	;
	791:L P[787] 200mm/sec CNT60 	;
	792:L P[788] 200mm/sec CNT60 	;
	793:L P[789] 200mm/sec CNT60 	;
	794:L P[790] 200mm/sec CNT60 	;
	795:L P[791] 200mm/sec CNT60 	;
	796:L P[792] 200mm/sec CNT60 	;
	797:L P[793] 200mm/sec CNT60 	;
	798:L P[794] 200mm/sec CNT60 	;
	799:L P[795] 200mm/sec CNT60 	;
	800:L P[796] 200mm/sec CNT60 	;
	801:L P[797] 200mm/sec CNT60 	;
	802:L P[798] 200mm/sec CNT60 	;
	803:L P[799] 200mm/sec CNT60 	;
	804:L P[800] 200mm/sec CNT60 	;
	805:L P[801] 200mm/sec CNT60 	;
	806:L P[802] 200mm/sec CNT60 	;
	807:L P[803] 200mm/sec CNT60 	;
	808:L P[804] 200mm/sec CNT60 	;
	809:L P[805] 200mm/sec CNT60 	;
	810:L P[806] 200mm/sec CNT60 	;
	811:L P[807] 200mm/sec CNT60 	;
	812:L P[808] 200mm/sec CNT60 	;
	813:L P[809] 200mm/sec CNT60 	;
	814:L P[810] 200mm/sec CNT60 	;
	815:L P[811] 200mm/sec CNT60 	;
	816:L P[812] 200mm/sec CNT60 	;
	817:L P[813] 200mm/sec CNT60 	;
	818:L P[814] 200mm/sec CNT60 	;
	819:L P[815] 200mm/sec CNT60 	;
	820:L P[816] 200mm/sec CNT60 	;
	821:L P[817] 200mm/sec CNT60 	;
	822:L P[818] 200mm/sec CNT60 	;
	823:L P[819] 200mm/sec CNT60 	;
	824:L P[820] 200mm/sec CNT60 	;
	825:L P[821] 200mm/sec CNT60 	;
	826:L P[822] 200mm/sec CNT60 	;
	827:L P[823] 200mm/sec CNT60 	;
	828:L P[824] 200mm/sec CNT60 	;
	829:L P[825] 200mm/sec CNT60 	;
	830:L P[826] 200mm/sec CNT60 	;
	831:L P[827] 200mm/sec CNT60 	;
	832:L P[828] 200mm/sec CNT60 	;
	833:L P[829] 200mm/sec CNT60 	;
	834:L P[830] 200mm/sec CNT60 	;
	835:L P[831] 200mm/sec CNT60 	;
	836:L P[832] 200mm/sec CNT60 	;
	837:L P[833] 200mm/sec CNT60 	;
	838:L P[834] 200mm/sec CNT60 	;
	839:L P[835] 200mm/sec CNT60 	;
	840:L P[836] 200mm/sec CNT60 	;
	841:L P[837] 200mm/sec CNT60 	;
	842:L P[838] 200mm/sec CNT60 	;
	843:L P[839] 200mm/sec CNT60 	;
	844:L P[840] 200mm/sec CNT60 	;
	845:L P[841] 200mm/sec CNT60 	;
	846:L P[842] 200mm/sec CNT60 	;
	847:L P[843] 200mm/sec CNT60 	;
	848:L P[844] 200mm/sec CNT60 	;
	849:L P[845] 200mm/sec CNT60 	;
	850:L P[846] 200mm/sec CNT60 	;
	851:L P[847] 200mm/sec CNT60 	;
	852:L P[848] 200mm/sec CNT60 	;
	853:L P[849] 200mm/sec CNT60 	;
	854:L P[850] 200mm/sec CNT60 	;
	855:L P[851] 200mm/sec CNT60 	;
	856:L P[852] 200mm/sec CNT60 	;
	857:L P[853] 200mm/sec CNT60 	;
	858:L P[854] 200mm/sec CNT60 	;
	859:L P[855] 200mm/sec CNT60 	;
	860:L P[856] 200mm/sec CNT60 	;
	861:L P[857] 200mm/sec CNT60 	;
	862:L P[858] 200mm/sec CNT60 	;
	863:L P[859] 200mm/sec CNT60 	;
	864:L P[860] 200mm/sec CNT60 	;
	865:L P[861] 200mm/sec CNT60 	;
	866:L P[862] 200mm/sec CNT60 	;
	867:L P[863] 200mm/sec CNT60 	;
	868:L P[864] 200mm/sec CNT60 	;
	869:L P[865] 200mm/sec CNT60 	;
	870:L P[866] 200mm/sec CNT60 	;
	871:L P[867] 200mm/sec CNT60 	;
	872:L P[868] 200mm/sec CNT60 	;
	873:L P[869] 200mm/sec CNT60 	;
	874:L P[870] 200mm/sec CNT60 	;
	875:L P[871] 200mm/sec CNT60 	;
	876:L P[872] 200mm/sec CNT60 	;
	877:L P[873] 200mm/sec CNT60 	;
	878:L P[874] 200mm/sec CNT60 	;
	879:L P[875] 200mm/sec CNT60 	;
	880:L P[876] 200mm/sec CNT60 	;
	881:L P[877] 200mm/sec CNT60 	;
	882:L P[878] 200mm/sec CNT60 	;
	883:L P[879] 200mm/sec CNT60 	;
	884:L P[880] 200mm/sec CNT60 	;
	885:L P[881] 200mm/sec CNT60 	;
	886:L P[882] 200mm/sec CNT60 	;
	887:L P[883] 200mm/sec CNT60 	;
	888:L P[884] 200mm/sec CNT60 	;
	889:L P[885] 200mm/sec CNT60 	;
	890:L P[886] 200mm/sec CNT60 	;
	891:L P[887] 200mm/sec CNT60 	;
	892:L P[888] 200mm/sec CNT60 	;
	893:L P[889] 200mm/sec CNT60 	;
	894:L P[890] 200mm/sec CNT60 	;
	895:L P[891] 200mm/sec CNT60 	;
	896:L P[892] 200mm/sec CNT60 	;
	897:L P[893] 200mm/sec CNT60 	;
	898:L P[894] 200mm/sec CNT60 	;
	899:L P[895] 200mm/sec CNT60 	;
	900:L P[896] 200mm/sec CNT60 	;
	901:L P[897] 200mm/sec CNT60 	;
	902:L P[898] 200mm/sec CNT60 	;
	903:L P[899] 200mm/sec CNT60 	;
	904:L P[900] 200mm/sec CNT60 	;
	905:L P[901] 200mm/sec CNT60 	;
	906:L P[902] 200mm/sec CNT60 	;
	907:L P[903] 200mm/sec CNT60 	;
	908:L P[904] 200mm/sec CNT60 	;
	909:L P[905] 200mm/sec CNT60 	;
	910:L P[906] 200mm/sec CNT60 	;
	911:L P[907] 200mm/sec CNT60 	;
	912:L P[908] 200mm/sec CNT60 	;
	913:L P[909] 200mm/sec CNT60 	;
/POS
P[1]{
   GP1:
	UF : 0, UT : 1,		CONFIG : 'N U T, 0, 0, 0',
	X =	1789.017057	mm,	Y =	678.561683	mm,	Z =	976.769836	mm,
	W =	-108.191512	deg,	P =	-49.248390	deg,	R =	71.820679	deg
};
P[2]{
   GP1:
	UF : 0, UT : 1,		CONFIG : 'N U T, 0, 0, 0',
	X =	1768.296777	mm,	Y =	691.589050	mm,	Z =	971.674975	mm,
	W =	-108.191512	deg,	P =	-49.248390	deg,	R =	71.820679	deg
};
P[3]{
   GP1:
	UF : 0, UT : 1,		CONFIG : 'N U T, 0, 0, 0',
	X =	1773.877759	mm,	Y =	698.766477	mm,	Z =	967.317055	mm,
	W =	-109.961961	deg,	P =	-50.186029	deg,	R =	71.470365	deg
};
P[4]{
   GP1:
	UF : 0, UT : 1,		CONFIG : 'N U T, 0, 0, 0',
	X =	1783.261711	mm,	Y =	709.958712	mm,	Z =	960.653642	mm,
	W =	-109.998091	deg,	P =	-51.120328	deg,	R =	70.000691	deg
};
P[5]{
   GP1:
	UF : 0, UT : 1,		CONFIG : 'N U T, 0, 0, 0',
	X =	1793.907059	mm,	Y =	722.084016	mm,	Z =	953.663000	mm,
	W =	-109.998091	deg,	P =	-51.120328	deg,	R =	70.000691	deg
};
P[6]{
   GP1:
	UF : 0, UT : 1,		CONFIG : 'N U T, 0, 0, 0',
	X =	1806.361780	mm,	Y =	735.764291	mm,	Z =	946.132376	mm,
	W =	-108.733496	deg,	P =	-27.818624	deg,	R =	59.882200	deg
};
P[7]{
   GP1:
	UF : 0, UT : 1,		CONFIG : 'N U T, 0, 0, 0',
	X =	1819.613062	mm,	Y =	748.791723	mm,	Z =	939.165517	mm,
	W =	-108.733496	deg,	P =	-27.818624	deg,	R =	59.882200	deg
};
P[8]{
   GP1:
	UF : 0, UT : 1,		CONFIG : 'N U T, 0, 0, 0',
	X =	1833.861613	mm,	Y =	761.785125	mm,	Z =	932.603056	mm,
	W =	-124.355697	deg,	P =	-54.122100	deg,	R =	74.297774	deg
};
P[9]{
   GP1:
	UF : 0, UT : 1,		CONFIG : 'N U T, 0, 0, 0',
	X =	1847.497419	mm,	Y =	772.946631	mm,	Z =	927.317076	mm,
	W =	-127.345217	deg,	P =	-55.364422	deg,	R =	74.344525	deg
};
P[10]{
   GP1:
	UF : 0, UT : 1,		CONFIG : 'N U T, 0, 0, 0',
	X =	1861.722854	mm,	Y =	783.572147	mm,	Z =	922.692799	mm,
	W =	-131.259404	deg,	P =	-56.468712	deg,	R =	75.059838	deg
};
P[11]{
   GP1:
	UF : 0, UT : 1,		CONFIG : 'N U T, 0, 0, 0',
	X =	1876.577070	mm,	Y =	793.577814	mm,	Z =	918.743989	mm,
	W =	-135.185777	deg,	P =	-57.929587	deg,	R =	75.465442	deg
};
P[12]{
   GP1:
	UF : 0, UT : 1,		CONFIG : 'N U T, 0, 0, 0',
	X =	1892.064953	mm,	Y =	802.866730	mm,	Z =	915.585118	mm,
	W =	-139.235996	deg,	P =	-59.375152	deg,	R =	76.051134	deg
};
P[13]{
   GP1:
	UF : 0, UT : 1,		CONFIG : 'N U T, 0, 0, 0',
	X =	1908.263374	mm,	Y =	811.505754	mm,	Z =	913.250873	mm,
	W =	-143.505255	deg,	P =	-59.928252	deg,	R =	77.546569	deg
};
P[14]{
   GP1:
	UF : 0, UT : 1,		CONFIG : 'N U T, 0, 0, 0',
	X =	1916.497449	mm,	Y =	815.468867	mm,	Z =	912.391724	mm,
	W =	-143.505255	deg,	P =	-59.928252	deg,	R =	77.546569	deg
};
P[15]{
   GP1:
	UF : 0, UT : 1,		CONFIG : 'N U T, 0, 0, 0',
	X =	1999.810179	mm,	Y =	834.921774	mm,	Z =	908.141556	mm,
	W =	-138.493937	deg,	P =	-50.635039	deg,	R =	44.709963	deg
};
P[16]{
   GP1:
	UF : 0, UT : 1,		CONFIG : 'N U T, 0, 0, 0',
	X =	1981.127687	mm,	Y =	832.016190	mm,	Z =	904.879371	mm,
	W =	-134.535792	deg,	P =	-47.752290	deg,	R =	46.215736	deg
};
P[17]{
   GP1:
	UF : 0, UT : 1,		CONFIG : 'N U T, 0, 0, 0',
	X =	1962.505798	mm,	Y =	827.614423	mm,	Z =	902.880165	mm,
	W =	-130.819033	deg,	P =	-45.448141	deg,	R =	47.316857	deg
};
P[18]{
   GP1:
	UF : 0, UT : 1,		CONFIG : 'N U T, 0, 0, 0',
	X =	1944.145300	mm,	Y =	821.998296	mm,	Z =	901.996165	mm,
	W =	-127.178740	deg,	P =	-42.820206	deg,	R =	48.793871	deg
};
P[19]{
   GP1:
	UF : 0, UT : 1,		CONFIG : 'N U T, 0, 0, 0',
	X =	1926.172765	mm,	Y =	815.104473	mm,	Z =	902.328312	mm,
	W =	-124.076141	deg,	P =	-40.298217	deg,	R =	50.402614	deg
};
P[20]{
   GP1:
	UF : 0, UT : 1,		CONFIG : 'N U T, 0, 0, 0',
	X =	1908.696350	mm,	Y =	807.052163	mm,	Z =	903.747133	mm,
	W =	-120.781033	deg,	P =	-38.287101	deg,	R =	51.461250	deg
};
P[21]{
   GP1:
	UF : 0, UT : 1,		CONFIG : 'N U T, 0, 0, 0',
	X =	1891.783336	mm,	Y =	798.078912	mm,	Z =	906.200751	mm,
	W =	-118.735346	deg,	P =	-35.964790	deg,	R =	53.366435	deg
};
P[22]{
   GP1:
	UF : 0, UT : 1,		CONFIG : 'N U T, 0, 0, 0',
	X =	1875.515159	mm,	Y =	788.235058	mm,	Z =	909.582937	mm,
	W =	-116.759942	deg,	P =	-33.742373	deg,	R =	55.289482	deg
};
P[23]{
   GP1:
	UF : 0, UT : 1,		CONFIG : 'N U T, 0, 0, 0',
	X =	1859.934398	mm,	Y =	777.566043	mm,	Z =	913.836539	mm,
	W =	-114.716321	deg,	P =	-32.011248	deg,	R =	56.677038	deg
};
P[24]{
   GP1:
	UF : 0, UT : 1,		CONFIG : 'N U T, 0, 0, 0',
	X =	1845.008105	mm,	Y =	766.253066	mm,	Z =	918.817565	mm,
	W =	-112.714831	deg,	P =	-30.523819	deg,	R =	57.824555	deg
};
P[25]{
   GP1:
	UF : 0, UT : 1,		CONFIG : 'N U T, 0, 0, 0',
	X =	1830.702871	mm,	Y =	754.399481	mm,	Z =	924.473343	mm,
	W =	-111.396961	deg,	P =	-29.248598	deg,	R =	59.013809	deg
};
P[26]{
   GP1:
	UF : 0, UT : 1,		CONFIG : 'N U T, 0, 0, 0',
	X =	1817.012560	mm,	Y =	742.204632	mm,	Z =	930.612328	mm,
	W =	-109.554532	deg,	P =	-27.294853	deg,	R =	61.014861	deg
};
P[27]{
   GP1:
	UF : 0, UT : 1,		CONFIG : 'N U T, 0, 0, 0',
	X =	1804.169109	mm,	Y =	729.354023	mm,	Z =	937.449141	mm,
	W =	-107.066264	deg,	P =	-26.263436	deg,	R =	61.433855	deg
};
P[28]{
   GP1:
	UF : 0, UT : 1,		CONFIG : 'N U T, 0, 0, 0',
	X =	1791.948185	mm,	Y =	716.080105	mm,	Z =	944.722285	mm,
	W =	-103.646321	deg,	P =	-25.705620	deg,	R =	60.562139	deg
};
P[29]{
   GP1:
	UF : 0, UT : 1,		CONFIG : 'N U T, 0, 0, 0',
	X =	1780.296108	mm,	Y =	702.680612	mm,	Z =	952.610573	mm,
	W =	-103.911926	deg,	P =	-24.236205	deg,	R =	63.096929	deg
};
P[30]{
   GP1:
	UF : 0, UT : 1,		CONFIG : 'N U T, 0, 0, 0',
	X =	1769.193539	mm,	Y =	688.841084	mm,	Z =	960.903744	mm,
	W =	-103.911926	deg,	P =	-24.236205	deg,	R =	63.096929	deg
};
P[31]{
   GP1:
	UF : 0, UT : 1,		CONFIG : 'N U T, 0, 0, 0',
	X =	1769.961995	mm,	Y =	685.878558	mm,	Z =	950.214570	mm,
	W =	-109.940294	deg,	P =	-49.662766	deg,	R =	72.312171	deg
};
P[32]{
   GP1:
	UF : 0, UT : 1,		CONFIG : 'N U T, 0, 0, 0',
	X =	1781.211184	mm,	Y =	699.748879	mm,	Z =	942.086217	mm,
	W =	-114.093092	deg,	P =	-49.997575	deg,	R =	74.380201	deg
};
P[33]{
   GP1:
	UF : 0, UT : 1,		CONFIG : 'N U T, 0, 0, 0',
	X =	1793.069370	mm,	Y =	713.201993	mm,	Z =	934.179196	mm,
	W =	-113.934983	deg,	P =	-51.831895	deg,	R =	71.489758	deg
};
P[34]{
   GP1:
	UF : 0, UT : 1,		CONFIG : 'N U T, 0, 0, 0',
	X =	1805.632332	mm,	Y =	726.409593	mm,	Z =	927.016620	mm,
	W =	-118.908089	deg,	P =	-52.189954	deg,	R =	73.911624	deg
};
P[35]{
   GP1:
	UF : 0, UT : 1,		CONFIG : 'N U T, 0, 0, 0',
	X =	1818.897863	mm,	Y =	739.180945	mm,	Z =	920.354072	mm,
	W =	-122.814290	deg,	P =	-52.843361	deg,	R =	75.120711	deg
};
P[36]{
   GP1:
	UF : 0, UT : 1,		CONFIG : 'N U T, 0, 0, 0',
	X =	1832.871942	mm,	Y =	751.495036	mm,	Z =	914.223284	mm,
	W =	-125.462914	deg,	P =	-53.681876	deg,	R =	75.400220	deg
};
P[37]{
   GP1:
	UF : 0, UT : 1,		CONFIG : 'N U T, 0, 0, 0',
	X =	1847.376358	mm,	Y =	763.368672	mm,	Z =	908.635375	mm,
	W =	-129.053026	deg,	P =	-54.674413	deg,	R =	75.969104	deg
};
P[38]{
   GP1:
	UF : 0, UT : 1,		CONFIG : 'N U T, 0, 0, 0',
	X =	1862.525801	mm,	Y =	774.635637	mm,	Z =	903.710656	mm,
	W =	-132.874887	deg,	P =	-56.184520	deg,	R =	76.122127	deg
};
P[39]{
   GP1:
	UF : 0, UT : 1,		CONFIG : 'N U T, 0, 0, 0',
	X =	1878.443973	mm,	Y =	785.176580	mm,	Z =	899.650952	mm,
	W =	-137.102554	deg,	P =	-57.449438	deg,	R =	76.804671	deg
};
P[40]{
   GP1:
	UF : 0, UT : 1,		CONFIG : 'N U T, 0, 0, 0',
	X =	1895.020521	mm,	Y =	794.954150	mm,	Z =	896.452010	mm,
	W =	-141.894227	deg,	P =	-58.520937	deg,	R =	77.966853	deg
};
P[41]{
   GP1:
	UF : 0, UT : 1,		CONFIG : 'N U T, 0, 0, 0',
	X =	1912.148400	mm,	Y =	803.865121	mm,	Z =	894.116658	mm,
	W =	-147.492388	deg,	P =	-60.088526	deg,	R =	79.158229	deg
};
P[42]{
   GP1:
	UF : 0, UT : 1,		CONFIG : 'N U T, 0, 0, 0',
	X =	1929.890036	mm,	Y =	811.701159	mm,	Z =	892.877020	mm,
	W =	-153.723441	deg,	P =	-61.550017	deg,	R =	80.847605	deg
};
P[43]{
   GP1:
	UF : 0, UT : 1,		CONFIG : 'N U T, 0, 0, 0',
	X =	1948.131247	mm,	Y =	818.388989	mm,	Z =	892.822042	mm,
	W =	-160.998722	deg,	P =	-62.185818	deg,	R =	83.469534	deg
};
P[44]{
   GP1:
	UF : 0, UT : 1,		CONFIG : 'N U T, 0, 0, 0',
	X =	1966.720329	mm,	Y =	823.861861	mm,	Z =	893.927627	mm,
	W =	-168.898684	deg,	P =	-62.335709	deg,	R =	86.381840	deg
};
P[45]{
   GP1:
	UF : 0, UT : 1,		CONFIG : 'N U T, 0, 0, 0',
	X =	1985.483943	mm,	Y =	827.965178	mm,	Z =	896.139790	mm,
	W =	-177.817793	deg,	P =	-63.594420	deg,	R =	89.468742	deg
};
P[46]{
   GP1:
	UF : 0, UT : 1,		CONFIG : 'N U T, 0, 0, 0',
	X =	2004.352706	mm,	Y =	830.470968	mm,	Z =	899.879523	mm,
	W =	174.199538	deg,	P =	-62.785824	deg,	R =	92.067568	deg
};
P[47]{
   GP1:
	UF : 0, UT : 1,		CONFIG : 'N U T, 0, 0, 0',
	X =	2023.061912	mm,	Y =	831.524250	mm,	Z =	904.725003	mm,
	W =	165.889324	deg,	P =	-62.668811	deg,	R =	94.573835	deg
};
P[48]{
   GP1:
	UF : 0, UT : 1,		CONFIG : 'N U T, 0, 0, 0',
	X =	2041.445422	mm,	Y =	830.988082	mm,	Z =	910.824495	mm,
	W =	158.986524	deg,	P =	-62.159974	deg,	R =	96.226989	deg
};
P[49]{
   GP1:
	UF : 0, UT : 1,		CONFIG : 'N U T, 0, 0, 0',
	X =	2059.768937	mm,	Y =	828.951581	mm,	Z =	918.029303	mm,
	W =	158.986524	deg,	P =	-62.159974	deg,	R =	96.226989	deg
};
P[50]{
   GP1:
	UF : 0, UT : 1,		CONFIG : 'N U T, 0, 0, 0',
	X =	2082.034497	mm,	Y =	819.885885	mm,	Z =	919.013592	mm,
	W =	150.718548	deg,	P =	-62.177184	deg,	R =	98.416508	deg
};
P[51]{
   GP1:
	UF : 0, UT : 1,		CONFIG : 'N U T, 0, 0, 0',
	X =	2064.585526	mm,	Y =	823.576434	mm,	Z =	910.681898	mm,
	W =	150.718548	deg,	P =	-62.177184	deg,	R =	98.416508	deg
};
P[52]{
   GP1:
	UF : 0, UT : 1,		CONFIG : 'N U T, 0, 0, 0',
	X =	2046.834552	mm,	Y =	825.876180	mm,	Z =	903.350309	mm,
	W =	157.189887	deg,	P =	-62.214632	deg,	R =	96.748325	deg
};
P[53]{
   GP1:
	UF : 0, UT : 1,		CONFIG : 'N U T, 0, 0, 0',
	X =	2028.588429	mm,	Y =	826.702426	mm,	Z =	897.115653	mm,
	W =	164.684739	deg,	P =	-62.002792	deg,	R =	94.589673	deg
};
P[54]{
   GP1:
	UF : 0, UT : 1,		CONFIG : 'N U T, 0, 0, 0',
	X =	2010.018180	mm,	Y =	826.047282	mm,	Z =	891.865463	mm,
	W =	171.875155	deg,	P =	-63.418470	deg,	R =	92.989573	deg
};
P[55]{
   GP1:
	UF : 0, UT : 1,		CONFIG : 'N U T, 0, 0, 0',
	X =	1991.241861	mm,	Y =	824.050088	mm,	Z =	887.804323	mm,
	W =	179.501315	deg,	P =	-63.484306	deg,	R =	90.413400	deg
};
P[56]{
   GP1:
	UF : 0, UT : 1,		CONFIG : 'N U T, 0, 0, 0',
	X =	1972.481014	mm,	Y =	820.542382	mm,	Z =	885.096905	mm,
	W =	-172.227017	deg,	P =	-62.371392	deg,	R =	87.552295	deg
};
P[57]{
   GP1:
	UF : 0, UT : 1,		CONFIG : 'N U T, 0, 0, 0',
	X =	1953.915673	mm,	Y =	815.526075	mm,	Z =	883.551355	mm,
	W =	-163.256176	deg,	P =	-62.828655	deg,	R =	84.124059	deg
};
P[58]{
   GP1:
	UF : 0, UT : 1,		CONFIG : 'N U T, 0, 0, 0',
	X =	1935.677333	mm,	Y =	809.194341	mm,	Z =	883.398670	mm,
	W =	-156.080138	deg,	P =	-61.154144	deg,	R =	82.006363	deg
};
P[59]{
   GP1:
	UF : 0, UT : 1,		CONFIG : 'N U T, 0, 0, 0',
	X =	1917.841385	mm,	Y =	801.710146	mm,	Z =	884.286057	mm,
	W =	-149.811801	deg,	P =	-60.100792	deg,	R =	80.110651	deg
};
P[60]{
   GP1:
	UF : 0, UT : 1,		CONFIG : 'N U T, 0, 0, 0',
	X =	1900.561151	mm,	Y =	793.179136	mm,	Z =	886.251793	mm,
	W =	-144.262506	deg,	P =	-58.673509	deg,	R =	78.845828	deg
};
P[61]{
   GP1:
	UF : 0, UT : 1,		CONFIG : 'N U T, 0, 0, 0',
	X =	1883.985371	mm,	Y =	783.624994	mm,	Z =	889.254324	mm,
	W =	-138.423433	deg,	P =	-57.430044	deg,	R =	77.406972	deg
};
P[62]{
   GP1:
	UF : 0, UT : 1,		CONFIG : 'N U T, 0, 0, 0',
	X =	1867.951221	mm,	Y =	773.322096	mm,	Z =	893.096488	mm,
	W =	-134.643286	deg,	P =	-56.136538	deg,	R =	76.973350	deg
};
P[63]{
   GP1:
	UF : 0, UT : 1,		CONFIG : 'N U T, 0, 0, 0',
	X =	1852.518995	mm,	Y =	762.366616	mm,	Z =	897.646386	mm,
	W =	-130.992797	deg,	P =	-55.088575	deg,	R =	76.414732	deg
};
P[64]{
   GP1:
	UF : 0, UT : 1,		CONFIG : 'N U T, 0, 0, 0',
	X =	1837.824913	mm,	Y =	750.779430	mm,	Z =	902.949340	mm,
	W =	-127.220681	deg,	P =	-53.911030	deg,	R =	75.981004	deg
};
P[65]{
   GP1:
	UF : 0, UT : 1,		CONFIG : 'N U T, 0, 0, 0',
	X =	1823.742493	mm,	Y =	738.688487	mm,	Z =	908.898360	mm,
	W =	-124.706265	deg,	P =	-52.698832	deg,	R =	76.250885	deg
};
P[66]{
   GP1:
	UF : 0, UT : 1,		CONFIG : 'N U T, 0, 0, 0',
	X =	1810.265570	mm,	Y =	726.139892	mm,	Z =	915.345055	mm,
	W =	-121.523734	deg,	P =	-51.996761	deg,	R =	75.575001	deg
};
P[67]{
   GP1:
	UF : 0, UT : 1,		CONFIG : 'N U T, 0, 0, 0',
	X =	1797.432825	mm,	Y =	713.226620	mm,	Z =	922.364420	mm,
	W =	-119.463095	deg,	P =	-50.871951	deg,	R =	76.062761	deg
};
P[68]{
   GP1:
	UF : 0, UT : 1,		CONFIG : 'N U T, 0, 0, 0',
	X =	1785.170537	mm,	Y =	699.936136	mm,	Z =	929.754307	mm,
	W =	-116.061589	deg,	P =	-50.472581	deg,	R =	74.794751	deg
};
P[69]{
   GP1:
	UF : 0, UT : 1,		CONFIG : 'N U T, 0, 0, 0',
	X =	1773.648267	mm,	Y =	686.296595	mm,	Z =	937.595668	mm,
	W =	-111.378941	deg,	P =	-50.083777	deg,	R =	72.567068	deg
};
P[70]{
   GP1:
	UF : 0, UT : 1,		CONFIG : 'N U T, 0, 0, 0',
	X =	1779.039000	mm,	Y =	688.119537	mm,	Z =	924.565464	mm,
	W =	-108.744771	deg,	P =	-24.955925	deg,	R =	64.227507	deg
};
P[71]{
   GP1:
	UF : 0, UT : 1,		CONFIG : 'N U T, 0, 0, 0',
	X =	1784.954000	mm,	Y =	694.814570	mm,	Z =	920.716666	mm,
	W =	-108.744771	deg,	P =	-24.955925	deg,	R =	64.227507	deg
};
P[72]{
   GP1:
	UF : 0, UT : 1,		CONFIG : 'N U T, 0, 0, 0',
	X =	1797.318334	mm,	Y =	708.140435	mm,	Z =	913.259840	mm,
	W =	-109.863550	deg,	P =	-25.646497	deg,	R =	63.620365	deg
};
P[73]{
   GP1:
	UF : 0, UT : 1,		CONFIG : 'N U T, 0, 0, 0',
	X =	1810.128362	mm,	Y =	721.079491	mm,	Z =	906.237667	mm,
	W =	-110.975232	deg,	P =	-26.663259	deg,	R =	62.539048	deg
};
P[74]{
   GP1:
	UF : 0, UT : 1,		CONFIG : 'N U T, 0, 0, 0',
	X =	1823.622462	mm,	Y =	733.534239	mm,	Z =	899.817064	mm,
	W =	-112.412068	deg,	P =	-28.182755	deg,	R =	60.912139	deg
};
P[75]{
   GP1:
	UF : 0, UT : 1,		CONFIG : 'N U T, 0, 0, 0',
	X =	1837.721329	mm,	Y =	745.615495	mm,	Z =	893.914359	mm,
	W =	-113.863406	deg,	P =	-29.430568	deg,	R =	59.743535	deg
};
P[76]{
   GP1:
	UF : 0, UT : 1,		CONFIG : 'N U T, 0, 0, 0',
	X =	1852.389180	mm,	Y =	757.256399	mm,	Z =	888.554727	mm,
	W =	-115.369135	deg,	P =	-30.726333	deg,	R =	58.579044	deg
};
P[77]{
   GP1:
	UF : 0, UT : 1,		CONFIG : 'N U T, 0, 0, 0',
	X =	1867.719451	mm,	Y =	768.247165	mm,	Z =	883.930067	mm,
	W =	-117.148004	deg,	P =	-32.517416	deg,	R =	56.937065	deg
};
P[78]{
   GP1:
	UF : 0, UT : 1,		CONFIG : 'N U T, 0, 0, 0',
	X =	1883.702122	mm,	Y =	778.573278	mm,	Z =	880.069696	mm,
	W =	-119.059071	deg,	P =	-34.338721	deg,	R =	55.387966	deg
};
P[79]{
   GP1:
	UF : 0, UT : 1,		CONFIG : 'N U T, 0, 0, 0',
	X =	1900.318975	mm,	Y =	788.111089	mm,	Z =	877.091977	mm,
	W =	-121.510640	deg,	P =	-36.272382	deg,	R =	53.961397	deg
};
P[80]{
   GP1:
	UF : 0, UT : 1,		CONFIG : 'N U T, 0, 0, 0',
	X =	1917.565219	mm,	Y =	796.645050	mm,	Z =	875.086921	mm,
	W =	-123.483677	deg,	P =	-38.857025	deg,	R =	51.746188	deg
};
P[81]{
   GP1:
	UF : 0, UT : 1,		CONFIG : 'N U T, 0, 0, 0',
	X =	1935.371531	mm,	Y =	804.094703	mm,	Z =	874.210757	mm,
	W =	-126.213408	deg,	P =	-41.442992	deg,	R =	49.890352	deg
};
P[82]{
   GP1:
	UF : 0, UT : 1,		CONFIG : 'N U T, 0, 0, 0',
	X =	1953.627035	mm,	Y =	810.480293	mm,	Z =	874.363919	mm,
	W =	-128.806432	deg,	P =	-43.887921	deg,	R =	48.230254	deg
};
P[83]{
   GP1:
	UF : 0, UT : 1,		CONFIG : 'N U T, 0, 0, 0',
	X =	1972.185229	mm,	Y =	815.678125	mm,	Z =	875.679414	mm,
	W =	-132.559144	deg,	P =	-46.158962	deg,	R =	47.139068	deg
};
P[84]{
   GP1:
	UF : 0, UT : 1,		CONFIG : 'N U T, 0, 0, 0',
	X =	1990.898457	mm,	Y =	819.275294	mm,	Z =	878.293579	mm,
	W =	-135.597241	deg,	P =	-49.698827	deg,	R =	44.764964	deg
};
P[85]{
   GP1:
	UF : 0, UT : 1,		CONFIG : 'N U T, 0, 0, 0',
	X =	2009.601935	mm,	Y =	821.322023	mm,	Z =	882.277026	mm,
	W =	-139.599187	deg,	P =	-52.830237	deg,	R =	43.138511	deg
};
P[86]{
   GP1:
	UF : 0, UT : 1,		CONFIG : 'N U T, 0, 0, 0',
	X =	2028.076627	mm,	Y =	821.865334	mm,	Z =	887.621913	mm,
	W =	-145.918331	deg,	P =	-54.749502	deg,	R =	43.080931	deg
};
P[87]{
   GP1:
	UF : 0, UT : 1,		CONFIG : 'N U T, 0, 0, 0',
	X =	2046.339928	mm,	Y =	821.009391	mm,	Z =	893.821754	mm,
	W =	-148.280037	deg,	P =	-57.797265	deg,	R =	41.292516	deg
};
P[88]{
   GP1:
	UF : 0, UT : 1,		CONFIG : 'N U T, 0, 0, 0',
	X =	2064.089931	mm,	Y =	818.892455	mm,	Z =	901.103427	mm,
	W =	-153.130525	deg,	P =	-59.629016	deg,	R =	40.961524	deg
};
P[89]{
   GP1:
	UF : 0, UT : 1,		CONFIG : 'N U T, 0, 0, 0',
	X =	2081.304750	mm,	Y =	815.488800	mm,	Z =	909.178950	mm,
	W =	-156.186271	deg,	P =	-62.203564	deg,	R =	39.815290	deg
};
P[90]{
   GP1:
	UF : 0, UT : 1,		CONFIG : 'N U T, 0, 0, 0',
	X =	2097.868568	mm,	Y =	810.984332	mm,	Z =	918.085532	mm,
	W =	-160.460216	deg,	P =	-63.807183	deg,	R =	39.529839	deg
};
P[91]{
   GP1:
	UF : 0, UT : 1,		CONFIG : 'N U T, 0, 0, 0',
	X =	2113.706393	mm,	Y =	805.512765	mm,	Z =	927.473790	mm,
	W =	-163.030186	deg,	P =	-65.894994	deg,	R =	38.737586	deg
};
P[92]{
   GP1:
	UF : 0, UT : 1,		CONFIG : 'N U T, 0, 0, 0',
	X =	2121.440362	mm,	Y =	802.333005	mm,	Z =	932.523729	mm,
	W =	-165.590045	deg,	P =	-67.537822	deg,	R =	38.247563	deg
};
P[93]{
   GP1:
	UF : 0, UT : 1,		CONFIG : 'N U T, 0, 0, 0',
	X =	2105.348346	mm,	Y =	813.148244	mm,	Z =	931.905866	mm,
	W =	140.579678	deg,	P =	-61.162511	deg,	R =	99.522784	deg
};
P[94]{
   GP1:
	UF : 0, UT : 1,		CONFIG : 'N U T, 0, 0, 0',
	X =	2102.641678	mm,	Y =	814.152175	mm,	Z =	930.251122	mm,
	W =	140.579678	deg,	P =	-61.162511	deg,	R =	99.522784	deg
};
P[95]{
   GP1:
	UF : 0, UT : 1,		CONFIG : 'N U T, 0, 0, 0',
	X =	2153.222151	mm,	Y =	781.209670	mm,	Z =	946.208066	mm,
	W =	126.270309	deg,	P =	-62.529285	deg,	R =	105.471584	deg
};
P[96]{
   GP1:
	UF : 0, UT : 1,		CONFIG : 'N U T, 0, 0, 0',
	X =	2139.151760	mm,	Y =	789.431119	mm,	Z =	935.084450	mm,
	W =	126.270309	deg,	P =	-62.529285	deg,	R =	105.471584	deg
};
P[97]{
   GP1:
	UF : 0, UT : 1,		CONFIG : 'N U T, 0, 0, 0',
	X =	2124.280531	mm,	Y =	796.547266	mm,	Z =	924.848765	mm,
	W =	135.098938	deg,	P =	-60.793792	deg,	R =	99.935078	deg
};
P[98]{
   GP1:
	UF : 0, UT : 1,		CONFIG : 'N U T, 0, 0, 0',
	X =	2108.697622	mm,	Y =	802.739265	mm,	Z =	914.948388	mm,
	W =	139.626657	deg,	P =	-60.578916	deg,	R =	98.823204	deg
};
P[99]{
   GP1:
	UF : 0, UT : 1,		CONFIG : 'N U T, 0, 0, 0',
	X =	2092.464501	mm,	Y =	807.929731	mm,	Z =	905.561593	mm,
	W =	143.317285	deg,	P =	-61.419235	deg,	R =	99.308178	deg
};
P[100]{
   GP1:
	UF : 0, UT : 1,		CONFIG : 'N U T, 0, 0, 0',
	X =	2075.532770	mm,	Y =	811.966944	mm,	Z =	896.980759	mm,
	W =	148.718043	deg,	P =	-61.831258	deg,	R =	98.558912	deg
};
P[101]{
   GP1:
	UF : 0, UT : 1,		CONFIG : 'N U T, 0, 0, 0',
	X =	2057.979057	mm,	Y =	814.949944	mm,	Z =	889.210537	mm,
	W =	154.586663	deg,	P =	-61.244840	deg,	R =	96.617034	deg
};
P[102]{
   GP1:
	UF : 0, UT : 1,		CONFIG : 'N U T, 0, 0, 0',
	X =	2039.968855	mm,	Y =	816.647067	mm,	Z =	882.192980	mm,
	W =	159.961394	deg,	P =	-62.396203	deg,	R =	96.120889	deg
};
P[103]{
   GP1:
	UF : 0, UT : 1,		CONFIG : 'N U T, 0, 0, 0',
	X =	2021.545951	mm,	Y =	817.015317	mm,	Z =	876.248413	mm,
	W =	166.808234	deg,	P =	-62.662847	deg,	R =	94.298205	deg
};
P[104]{
   GP1:
	UF : 0, UT : 1,		CONFIG : 'N U T, 0, 0, 0',
	X =	2002.844782	mm,	Y =	815.876416	mm,	Z =	871.504093	mm,
	W =	174.713990	deg,	P =	-62.547774	deg,	R =	91.851699	deg
};
P[105]{
   GP1:
	UF : 0, UT : 1,		CONFIG : 'N U T, 0, 0, 0',
	X =	1984.052317	mm,	Y =	813.130615	mm,	Z =	868.123201	mm,
	W =	-176.790369	deg,	P =	-61.731750	deg,	R =	89.108449	deg
};
P[106]{
   GP1:
	UF : 0, UT : 1,		CONFIG : 'N U T, 0, 0, 0',
	X =	1965.339669	mm,	Y =	808.856084	mm,	Z =	866.018720	mm,
	W =	-168.699653	deg,	P =	-61.136179	deg,	R =	86.563386	deg
};
P[107]{
   GP1:
	UF : 0, UT : 1,		CONFIG : 'N U T, 0, 0, 0',
	X =	1946.865284	mm,	Y =	803.189164	mm,	Z =	865.103565	mm,
	W =	-160.762219	deg,	P =	-61.008053	deg,	R =	83.843992	deg
};
P[108]{
   GP1:
	UF : 0, UT : 1,		CONFIG : 'N U T, 0, 0, 0',
	X =	1928.658307	mm,	Y =	796.446498	mm,	Z =	865.268933	mm,
	W =	-154.918924	deg,	P =	-60.026714	deg,	R =	82.147575	deg
};
P[109]{
   GP1:
	UF : 0, UT : 1,		CONFIG : 'N U T, 0, 0, 0',
	X =	1911.100985	mm,	Y =	788.446187	mm,	Z =	866.698438	mm,
	W =	-148.243255	deg,	P =	-58.494999	deg,	R =	80.565411	deg
};
P[110]{
   GP1:
	UF : 0, UT : 1,		CONFIG : 'N U T, 0, 0, 0',
	X =	1894.037988	mm,	Y =	779.469920	mm,	Z =	869.104483	mm,
	W =	-143.325362	deg,	P =	-57.208172	deg,	R =	79.626105	deg
};
P[111]{
   GP1:
	UF : 0, UT : 1,		CONFIG : 'N U T, 0, 0, 0',
	X =	1877.554248	mm,	Y =	769.650073	mm,	Z =	872.355646	mm,
	W =	-138.532738	deg,	P =	-56.313973	deg,	R =	78.470408	deg
};
P[112]{
   GP1:
	UF : 0, UT : 1,		CONFIG : 'N U T, 0, 0, 0',
	X =	1861.794161	mm,	Y =	759.034934	mm,	Z =	876.510149	mm,
	W =	-133.917164	deg,	P =	-55.143352	deg,	R =	77.661160	deg
};
P[113]{
   GP1:
	UF : 0, UT : 1,		CONFIG : 'N U T, 0, 0, 0',
	X =	1846.647309	mm,	Y =	747.782356	mm,	Z =	881.421777	mm,
	W =	-130.655653	deg,	P =	-53.912738	deg,	R =	77.557858	deg
};
P[114]{
   GP1:
	UF : 0, UT : 1,		CONFIG : 'N U T, 0, 0, 0',
	X =	1832.171224	mm,	Y =	735.956957	mm,	Z =	887.008936	mm,
	W =	-127.528191	deg,	P =	-52.775037	deg,	R =	77.480603	deg
};
P[115]{
   GP1:
	UF : 0, UT : 1,		CONFIG : 'N U T, 0, 0, 0',
	X =	1818.363709	mm,	Y =	723.622684	mm,	Z =	893.203817	mm,
	W =	-124.392409	deg,	P =	-51.833727	deg,	R =	77.204819	deg
};
P[116]{
   GP1:
	UF : 0, UT : 1,		CONFIG : 'N U T, 0, 0, 0',
	X =	1805.089265	mm,	Y =	710.899498	mm,	Z =	899.893405	mm,
	W =	-122.010624	deg,	P =	-51.058068	deg,	R =	77.090295	deg
};
P[117]{
   GP1:
	UF : 0, UT : 1,		CONFIG : 'N U T, 0, 0, 0',
	X =	1792.351197	mm,	Y =	697.859962	mm,	Z =	907.046688	mm,
	W =	-120.328813	deg,	P =	-50.132195	deg,	R =	77.556822	deg
};
P[118]{
   GP1:
	UF : 0, UT : 1,		CONFIG : 'N U T, 0, 0, 0',
	X =	1780.239929	mm,	Y =	684.493227	mm,	Z =	914.620133	mm,
	W =	-117.930551	deg,	P =	-49.377833	deg,	R =	77.456225	deg
};
P[119]{
   GP1:
	UF : 0, UT : 1,		CONFIG : 'N U T, 0, 0, 0',
	X =	1778.650204	mm,	Y =	677.525449	mm,	Z =	906.634714	mm,
	W =	-109.793793	deg,	P =	-24.818499	deg,	R =	64.877698	deg
};
P[120]{
   GP1:
	UF : 0, UT : 1,		CONFIG : 'N U T, 0, 0, 0',
	X =	1784.688375	mm,	Y =	684.311937	mm,	Z =	902.746032	mm,
	W =	-109.793793	deg,	P =	-24.818499	deg,	R =	64.877698	deg
};
P[121]{
   GP1:
	UF : 0, UT : 1,		CONFIG : 'N U T, 0, 0, 0',
	X =	1790.928494	mm,	Y =	691.077829	mm,	Z =	898.935045	mm,
	W =	-110.394231	deg,	P =	-25.366108	deg,	R =	64.265167	deg
};
P[122]{
   GP1:
	UF : 0, UT : 1,		CONFIG : 'N U T, 0, 0, 0',
	X =	1803.735289	mm,	Y =	704.340397	mm,	Z =	891.646760	mm,
	W =	-111.281235	deg,	P =	-26.063042	deg,	R =	63.553020	deg
};
P[123]{
   GP1:
	UF : 0, UT : 1,		CONFIG : 'N U T, 0, 0, 0',
	X =	1817.058180	mm,	Y =	717.258583	mm,	Z =	884.818539	mm,
	W =	-112.695115	deg,	P =	-27.052258	deg,	R =	62.632185	deg
};
P[124]{
   GP1:
	UF : 0, UT : 1,		CONFIG : 'N U T, 0, 0, 0',
	X =	1830.960640	mm,	Y =	729.774560	mm,	Z =	878.466458	mm,
	W =	-113.840453	deg,	P =	-28.309421	deg,	R =	61.272092	deg
};
P[125]{
   GP1:
	UF : 0, UT : 1,		CONFIG : 'N U T, 0, 0, 0',
	X =	1845.573330	mm,	Y =	741.723381	mm,	Z =	872.832784	mm,
	W =	-115.720361	deg,	P =	-29.918683	deg,	R =	59.762747	deg
};
P[126]{
   GP1:
	UF : 0, UT : 1,		CONFIG : 'N U T, 0, 0, 0',
	X =	1860.860500	mm,	Y =	753.126210	mm,	Z =	867.866021	mm,
	W =	-117.576982	deg,	P =	-31.456826	deg,	R =	58.411593	deg
};
P[127]{
   GP1:
	UF : 0, UT : 1,		CONFIG : 'N U T, 0, 0, 0',
	X =	1876.768113	mm,	Y =	763.932348	mm,	Z =	863.562310	mm,
	W =	-119.128411	deg,	P =	-33.116768	deg,	R =	56.874493	deg
};
P[128]{
   GP1:
	UF : 0, UT : 1,		CONFIG : 'N U T, 0, 0, 0',
	X =	1893.335569	mm,	Y =	773.936126	mm,	Z =	860.139073	mm,
	W =	-121.128947	deg,	P =	-35.190442	deg,	R =	55.072896	deg
};
P[129]{
   GP1:
	UF : 0, UT : 1,		CONFIG : 'N U T, 0, 0, 0',
	X =	1910.536660	mm,	Y =	783.094503	mm,	Z =	857.723375	mm,
	W =	-124.542884	deg,	P =	-36.930756	deg,	R =	54.153244	deg
};
P[130]{
   GP1:
	UF : 0, UT : 1,		CONFIG : 'N U T, 0, 0, 0',
	X =	1928.315051	mm,	Y =	791.273573	mm,	Z =	856.262889	mm,
	W =	-127.543102	deg,	P =	-38.953617	deg,	R =	52.832615	deg
};
P[131]{
   GP1:
	UF : 0, UT : 1,		CONFIG : 'N U T, 0, 0, 0',
	X =	1946.616709	mm,	Y =	798.143416	mm,	Z =	855.997121	mm,
	W =	-130.250600	deg,	P =	-41.926609	deg,	R =	50.553639	deg
};
P[132]{
   GP1:
	UF : 0, UT : 1,		CONFIG : 'N U T, 0, 0, 0',
	X =	1965.330663	mm,	Y =	803.818053	mm,	Z =	856.895087	mm,
	W =	-133.215822	deg,	P =	-44.527892	deg,	R =	48.827347	deg
};
P[133]{
   GP1:
	UF : 0, UT : 1,		CONFIG : 'N U T, 0, 0, 0',
	X =	1984.274175	mm,	Y =	808.121057	mm,	Z =	859.022683	mm,
	W =	-136.475514	deg,	P =	-47.347385	deg,	R =	47.067984	deg
};
P[134]{
   GP1:
	UF : 0, UT : 1,		CONFIG : 'N U T, 0, 0, 0',
	X =	2003.265118	mm,	Y =	811.004135	mm,	Z =	862.521784	mm,
	W =	-142.036304	deg,	P =	-49.294342	deg,	R =	46.616167	deg
};
P[135]{
   GP1:
	UF : 0, UT : 1,		CONFIG : 'N U T, 0, 0, 0',
	X =	2022.125500	mm,	Y =	812.067249	mm,	Z =	867.238874	mm,
	W =	-144.426747	deg,	P =	-53.511582	deg,	R =	43.726217	deg
};
P[136]{
   GP1:
	UF : 0, UT : 1,		CONFIG : 'N U T, 0, 0, 0',
	X =	2040.690543	mm,	Y =	811.625346	mm,	Z =	873.233859	mm,
	W =	-147.877550	deg,	P =	-56.689325	deg,	R =	42.026858	deg
};
P[137]{
   GP1:
	UF : 0, UT : 1,		CONFIG : 'N U T, 0, 0, 0',
	X =	2058.917629	mm,	Y =	810.060182	mm,	Z =	880.284349	mm,
	W =	-153.580231	deg,	P =	-57.522814	deg,	R =	42.457668	deg
};
P[138]{
   GP1:
	UF : 0, UT : 1,		CONFIG : 'N U T, 0, 0, 0',
	X =	2076.494627	mm,	Y =	806.935354	mm,	Z =	888.205862	mm,
	W =	-156.632573	deg,	P =	-60.774804	deg,	R =	40.795517	deg
};
P[139]{
   GP1:
	UF : 0, UT : 1,		CONFIG : 'N U T, 0, 0, 0',
	X =	2093.562993	mm,	Y =	802.678643	mm,	Z =	896.897270	mm,
	W =	-158.751280	deg,	P =	-63.465852	deg,	R =	39.469178	deg
};
P[140]{
   GP1:
	UF : 0, UT : 1,		CONFIG : 'N U T, 0, 0, 0',
	X =	2110.072487	mm,	Y =	797.603918	mm,	Z =	906.318020	mm,
	W =	-163.126732	deg,	P =	-64.039695	deg,	R =	39.737328	deg
};
P[141]{
   GP1:
	UF : 0, UT : 1,		CONFIG : 'N U T, 0, 0, 0',
	X =	2125.741314	mm,	Y =	791.306991	mm,	Z =	916.270893	mm,
	W =	-165.186030	deg,	P =	-67.192265	deg,	R =	38.363542	deg
};
P[142]{
   GP1:
	UF : 0, UT : 1,		CONFIG : 'N U T, 0, 0, 0',
	X =	2140.789966	mm,	Y =	784.195718	mm,	Z =	926.782588	mm,
	W =	-167.422472	deg,	P =	-69.120479	deg,	R =	37.751416	deg
};
P[143]{
   GP1:
	UF : 0, UT : 1,		CONFIG : 'N U T, 0, 0, 0',
	X =	2154.885698	mm,	Y =	776.244604	mm,	Z =	937.903348	mm,
	W =	-172.150643	deg,	P =	-69.922673	deg,	R =	37.886426	deg
};
P[144]{
   GP1:
	UF : 0, UT : 1,		CONFIG : 'N U T, 0, 0, 0',
	X =	2168.248186	mm,	Y =	767.251205	mm,	Z =	949.198864	mm,
	W =	-171.798687	deg,	P =	-74.407258	deg,	R =	36.436816	deg
};
P[145]{
   GP1:
	UF : 0, UT : 1,		CONFIG : 'N U T, 0, 0, 0',
	X =	2180.587638	mm,	Y =	757.608956	mm,	Z =	961.069265	mm,
	W =	-175.446834	deg,	P =	-76.227068	deg,	R =	36.670902	deg
};
P[146]{
   GP1:
	UF : 0, UT : 1,		CONFIG : 'N U T, 0, 0, 0',
	X =	2202.785974	mm,	Y =	735.480321	mm,	Z =	972.903465	mm,
	W =	117.481330	deg,	P =	-61.688819	deg,	R =	105.481847	deg
};
P[147]{
   GP1:
	UF : 0, UT : 1,		CONFIG : 'N U T, 0, 0, 0',
	X =	2190.761088	mm,	Y =	745.562191	mm,	Z =	960.830850	mm,
	W =	117.481330	deg,	P =	-61.688819	deg,	R =	105.481847	deg
};
P[148]{
   GP1:
	UF : 0, UT : 1,		CONFIG : 'N U T, 0, 0, 0',
	X =	2178.632505	mm,	Y =	755.538809	mm,	Z =	948.813649	mm,
	W =	118.085768	deg,	P =	-61.675517	deg,	R =	105.298917	deg
};
P[149]{
   GP1:
	UF : 0, UT : 1,		CONFIG : 'N U T, 0, 0, 0',
	X =	2165.954239	mm,	Y =	764.898846	mm,	Z =	937.119097	mm,
	W =	121.166976	deg,	P =	-61.704843	deg,	R =	104.685549	deg
};
P[150]{
   GP1:
	UF : 0, UT : 1,		CONFIG : 'N U T, 0, 0, 0',
	X =	2152.311531	mm,	Y =	773.427758	mm,	Z =	926.079128	mm,
	W =	129.470586	deg,	P =	-60.045603	deg,	R =	99.151749	deg
};
P[151]{
   GP1:
	UF : 0, UT : 1,		CONFIG : 'N U T, 0, 0, 0',
	X =	2137.880274	mm,	Y =	780.986852	mm,	Z =	915.280033	mm,
	W =	132.960718	deg,	P =	-60.455011	deg,	R =	99.624878	deg
};
P[152]{
   GP1:
	UF : 0, UT : 1,		CONFIG : 'N U T, 0, 0, 0',
	X =	2122.731950	mm,	Y =	787.888993	mm,	Z =	904.968174	mm,
	W =	137.392273	deg,	P =	-59.859166	deg,	R =	97.983228	deg
};
P[153]{
   GP1:
	UF : 0, UT : 1,		CONFIG : 'N U T, 0, 0, 0',
	X =	2106.858595	mm,	Y =	793.746849	mm,	Z =	895.244858	mm,
	W =	142.281160	deg,	P =	-59.637116	deg,	R =	97.057897	deg
};
P[154]{
   GP1:
	UF : 0, UT : 1,		CONFIG : 'N U T, 0, 0, 0',
	X =	2090.391661	mm,	Y =	798.742706	mm,	Z =	885.926565	mm,
	W =	145.065649	deg,	P =	-60.731727	deg,	R =	98.070608	deg
};
P[155]{
   GP1:
	UF : 0, UT : 1,		CONFIG : 'N U T, 0, 0, 0',
	X =	2073.308214	mm,	Y =	802.766949	mm,	Z =	877.384049	mm,
	W =	150.100480	deg,	P =	-60.521866	deg,	R =	96.881819	deg
};
P[156]{
   GP1:
	UF : 0, UT : 1,		CONFIG : 'N U T, 0, 0, 0',
	X =	2055.613366	mm,	Y =	805.342879	mm,	Z =	869.794645	mm,
	W =	156.529043	deg,	P =	-60.820240	deg,	R =	95.839584	deg
};
P[157]{
   GP1:
	UF : 0, UT : 1,		CONFIG : 'N U T, 0, 0, 0',
	X =	2037.391917	mm,	Y =	806.772531	mm,	Z =	863.035536	mm,
	W =	162.044265	deg,	P =	-61.012197	deg,	R =	94.720450	deg
};
P[158]{
   GP1:
	UF : 0, UT : 1,		CONFIG : 'N U T, 0, 0, 0',
	X =	2018.813666	mm,	Y =	806.941524	mm,	Z =	857.228568	mm,
	W =	168.125978	deg,	P =	-61.114706	deg,	R =	93.279375	deg
};
P[159]{
   GP1:
	UF : 0, UT : 1,		CONFIG : 'N U T, 0, 0, 0',
	X =	2000.004724	mm,	Y =	805.526718	mm,	Z =	852.794880	mm,
	W =	176.032164	deg,	P =	-59.686874	deg,	R =	90.941962	deg
};
P[160]{
   GP1:
	UF : 0, UT : 1,		CONFIG : 'N U T, 0, 0, 0',
	X =	1981.179734	mm,	Y =	802.341076	mm,	Z =	849.640935	mm,
	W =	-175.342803	deg,	P =	-60.164384	deg,	R =	88.731202	deg
};
P[161]{
   GP1:
	UF : 0, UT : 1,		CONFIG : 'N U T, 0, 0, 0',
	X =	1962.426236	mm,	Y =	797.719243	mm,	Z =	847.725261	mm,
	W =	-167.391943	deg,	P =	-60.574503	deg,	R =	86.265531	deg
};
P[162]{
   GP1:
	UF : 0, UT : 1,		CONFIG : 'N U T, 0, 0, 0',
	X =	1943.863559	mm,	Y =	791.911191	mm,	Z =	846.981035	mm,
	W =	-160.986779	deg,	P =	-59.803316	deg,	R =	84.406312	deg
};
P[163]{
   GP1:
	UF : 0, UT : 1,		CONFIG : 'N U T, 0, 0, 0',
	X =	1925.773407	mm,	Y =	784.850744	mm,	Z =	847.553614	mm,
	W =	-155.303774	deg,	P =	-57.557864	deg,	R =	83.617470	deg
};
P[164]{
   GP1:
	UF : 0, UT : 1,		CONFIG : 'N U T, 0, 0, 0',
	X =	1908.174606	mm,	Y =	776.655859	mm,	Z =	849.112672	mm,
	W =	-149.674802	deg,	P =	-56.580916	deg,	R =	82.389039	deg
};
P[165]{
   GP1:
	UF : 0, UT : 1,		CONFIG : 'N U T, 0, 0, 0',
	X =	1891.138906	mm,	Y =	767.458433	mm,	Z =	851.521246	mm,
	W =	-142.689743	deg,	P =	-57.058381	deg,	R =	79.498517	deg
};
P[166]{
   GP1:
	UF : 0, UT : 1,		CONFIG : 'N U T, 0, 0, 0',
	X =	1874.786613	mm,	Y =	757.477818	mm,	Z =	855.161570	mm,
	W =	-140.104708	deg,	P =	-54.239545	deg,	R =	80.970186	deg
};
P[167]{
   GP1:
	UF : 0, UT : 1,		CONFIG : 'N U T, 0, 0, 0',
	X =	1859.115962	mm,	Y =	746.612596	mm,	Z =	859.422557	mm,
	W =	-134.192592	deg,	P =	-54.255132	deg,	R =	78.694011	deg
};
P[168]{
   GP1:
	UF : 0, UT : 1,		CONFIG : 'N U T, 0, 0, 0',
	X =	1844.012144	mm,	Y =	735.207948	mm,	Z =	864.478603	mm,
	W =	-131.253122	deg,	P =	-53.119949	deg,	R =	78.699480	deg
};
P[169]{
   GP1:
	UF : 0, UT : 1,		CONFIG : 'N U T, 0, 0, 0',
	X =	1829.632186	mm,	Y =	723.237030	mm,	Z =	870.232673	mm,
	W =	-128.260954	deg,	P =	-51.879730	deg,	R =	78.881156	deg
};
P[170]{
   GP1:
	UF : 0, UT : 1,		CONFIG : 'N U T, 0, 0, 0',
	X =	1815.777143	mm,	Y =	710.802281	mm,	Z =	876.465758	mm,
	W =	-125.208312	deg,	P =	-51.368372	deg,	R =	78.181464	deg
};
P[171]{
   GP1:
	UF : 0, UT : 1,		CONFIG : 'N U T, 0, 0, 0',
	X =	1802.587914	mm,	Y =	697.987282	mm,	Z =	883.292408	mm,
	W =	-122.970179	deg,	P =	-50.289777	deg,	R =	78.592896	deg
};
P[172]{
   GP1:
	UF : 0, UT : 1,		CONFIG : 'N U T, 0, 0, 0',
	X =	1790.046491	mm,	Y =	684.807635	mm,	Z =	890.569764	mm,
	W =	-120.290234	deg,	P =	-49.575147	deg,	R =	78.339620	deg
};
P[173]{
   GP1:
	UF : 0, UT : 1,		CONFIG : 'N U T, 0, 0, 0',
	X =	1783.880413	mm,	Y =	678.106386	mm,	Z =	894.354402	mm,
	W =	-119.363558	deg,	P =	-49.146199	deg,	R =	78.520196	deg
};
P[174]{
   GP1:
	UF : 0, UT : 1,		CONFIG : 'N U T, 0, 0, 0',
	X =	1785.430401	mm,	Y =	674.495792	mm,	Z =	884.489525	mm,
	W =	-111.522113	deg,	P =	-25.428066	deg,	R =	64.604004	deg
};
P[175]{
   GP1:
	UF : 0, UT : 1,		CONFIG : 'N U T, 0, 0, 0',
	X =	1798.065974	mm,	Y =	687.943331	mm,	Z =	876.985256	mm,
	W =	-111.522113	deg,	P =	-25.428066	deg,	R =	64.604004	deg
};
P[176]{
   GP1:
	UF : 0, UT : 1,		CONFIG : 'N U T, 0, 0, 0',
	X =	1811.172163	mm,	Y =	700.990964	mm,	Z =	869.999475	mm,
	W =	-113.143064	deg,	P =	-26.361173	deg,	R =	63.799085	deg
};
P[177]{
   GP1:
	UF : 0, UT : 1,		CONFIG : 'N U T, 0, 0, 0',
	X =	1824.829451	mm,	Y =	713.678625	mm,	Z =	863.427134	mm,
	W =	-114.177360	deg,	P =	-27.505485	deg,	R =	62.517026	deg
};
P[178]{
   GP1:
	UF : 0, UT : 1,		CONFIG : 'N U T, 0, 0, 0',
	X =	1839.143930	mm,	Y =	725.882833	mm,	Z =	857.516016	mm,
	W =	-116.211891	deg,	P =	-28.817426	deg,	R =	61.396057	deg
};
P[179]{
   GP1:
	UF : 0, UT : 1,		CONFIG : 'N U T, 0, 0, 0',
	X =	1854.089103	mm,	Y =	737.570780	mm,	Z =	852.116690	mm,
	W =	-116.893872	deg,	P =	-30.504670	deg,	R =	59.398444	deg
};
P[180]{
   GP1:
	UF : 0, UT : 1,		CONFIG : 'N U T, 0, 0, 0',
	X =	1869.718494	mm,	Y =	748.656394	mm,	Z =	847.653635	mm,
	W =	-120.534046	deg,	P =	-31.712635	deg,	R =	59.014521	deg
};
P[181]{
   GP1:
	UF : 0, UT : 1,		CONFIG : 'N U T, 0, 0, 0',
	X =	1886.039435	mm,	Y =	758.962004	mm,	Z =	843.910609	mm,
	W =	-122.587665	deg,	P =	-33.590130	deg,	R =	57.359619	deg
};
P[182]{
   GP1:
	UF : 0, UT : 1,		CONFIG : 'N U T, 0, 0, 0',
	X =	1902.960514	mm,	Y =	768.556790	mm,	Z =	840.958257	mm,
	W =	-124.683360	deg,	P =	-35.331329	deg,	R =	55.952669	deg
};
P[183]{
   GP1:
	UF : 0, UT : 1,		CONFIG : 'N U T, 0, 0, 0',
	X =	1920.496212	mm,	Y =	777.089664	mm,	Z =	839.056130	mm,
	W =	-126.999211	deg,	P =	-37.861420	deg,	R =	53.829034	deg
};
P[184]{
   GP1:
	UF : 0, UT : 1,		CONFIG : 'N U T, 0, 0, 0',
	X =	1938.588076	mm,	Y =	784.551766	mm,	Z =	838.260263	mm,
	W =	-129.806599	deg,	P =	-40.272933	deg,	R =	52.075056	deg
};
P[185]{
   GP1:
	UF : 0, UT : 1,		CONFIG : 'N U T, 0, 0, 0',
	X =	1957.112147	mm,	Y =	790.933229	mm,	Z =	838.581100	mm,
	W =	-133.558277	deg,	P =	-42.215443	deg,	R =	51.074821	deg
};
P[186]{
   GP1:
	UF : 0, UT : 1,		CONFIG : 'N U T, 0, 0, 0',
	X =	1975.927158	mm,	Y =	795.802330	mm,	Z =	840.231772	mm,
	W =	-137.564159	deg,	P =	-45.040332	deg,	R =	49.346177	deg
};
P[187]{
   GP1:
	UF : 0, UT : 1,		CONFIG : 'N U T, 0, 0, 0',
	X =	1994.911479	mm,	Y =	799.305519	mm,	Z =	843.176194	mm,
	W =	-142.564864	deg,	P =	-47.004949	deg,	R =	48.585821	deg
};
P[188]{
   GP1:
	UF : 0, UT : 1,		CONFIG : 'N U T, 0, 0, 0',
	X =	2013.963799	mm,	Y =	801.342158	mm,	Z =	847.064973	mm,
	W =	-143.549153	deg,	P =	-50.827590	deg,	R =	45.670100	deg
};
P[189]{
   GP1:
	UF : 0, UT : 1,		CONFIG : 'N U T, 0, 0, 0',
	X =	2032.704844	mm,	Y =	801.962135	mm,	Z =	852.439954	mm,
	W =	-149.800450	deg,	P =	-52.439497	deg,	R =	45.469757	deg
};
P[190]{
   GP1:
	UF : 0, UT : 1,		CONFIG : 'N U T, 0, 0, 0',
	X =	2051.054940	mm,	Y =	800.741606	mm,	Z =	858.843348	mm,
	W =	-151.240114	deg,	P =	-57.190871	deg,	R =	42.307692	deg
};
P[191]{
   GP1:
	UF : 0, UT : 1,		CONFIG : 'N U T, 0, 0, 0',
	X =	2068.984048	mm,	Y =	798.375015	mm,	Z =	866.361069	mm,
	W =	-155.496164	deg,	P =	-58.977212	deg,	R =	41.777578	deg
};
P[192]{
   GP1:
	UF : 0, UT : 1,		CONFIG : 'N U T, 0, 0, 0',
	X =	2086.427163	mm,	Y =	794.872114	mm,	Z =	874.632910	mm,
	W =	-158.823132	deg,	P =	-60.847362	deg,	R =	41.052726	deg
};
P[193]{
   GP1:
	UF : 0, UT : 1,		CONFIG : 'N U T, 0, 0, 0',
	X =	2103.111661	mm,	Y =	790.114972	mm,	Z =	883.703282	mm,
	W =	-162.163284	deg,	P =	-63.316106	deg,	R =	40.023300	deg
};
P[194]{
   GP1:
	UF : 0, UT : 1,		CONFIG : 'N U T, 0, 0, 0',
	X =	2119.115738	mm,	Y =	784.329325	mm,	Z =	893.483749	mm,
	W =	-165.759844	deg,	P =	-64.943296	deg,	R =	39.523983	deg
};
P[195]{
   GP1:
	UF : 0, UT : 1,		CONFIG : 'N U T, 0, 0, 0',
	X =	2134.632392	mm,	Y =	777.755184	mm,	Z =	903.703244	mm,
	W =	-167.888024	deg,	P =	-66.457277	deg,	R =	38.977169	deg
};
P[196]{
   GP1:
	UF : 0, UT : 1,		CONFIG : 'N U T, 0, 0, 0',
	X =	2149.365394	mm,	Y =	770.335037	mm,	Z =	914.409274	mm,
	W =	-170.532455	deg,	P =	-68.283463	deg,	R =	38.384637	deg
};
P[197]{
   GP1:
	UF : 0, UT : 1,		CONFIG : 'N U T, 0, 0, 0',
	X =	2163.511747	mm,	Y =	762.135209	mm,	Z =	925.421382	mm,
	W =	-171.113325	deg,	P =	-71.109133	deg,	R =	37.398911	deg
};
P[198]{
   GP1:
	UF : 0, UT : 1,		CONFIG : 'N U T, 0, 0, 0',
	X =	2176.660760	mm,	Y =	753.205504	mm,	Z =	936.963595	mm,
	W =	-174.616477	deg,	P =	-72.731972	deg,	R =	37.238556	deg
};
P[199]{
   GP1:
	UF : 0, UT : 1,		CONFIG : 'N U T, 0, 0, 0',
	X =	2188.975749	mm,	Y =	743.398802	mm,	Z =	948.759060	mm,
	W =	-176.047249	deg,	P =	-76.110929	deg,	R =	36.782393	deg
};
P[200]{
   GP1:
	UF : 0, UT : 1,		CONFIG : 'N U T, 0, 0, 0',
	X =	2200.903684	mm,	Y =	733.340788	mm,	Z =	960.968518	mm,
	W =	-178.877336	deg,	P =	-75.592772	deg,	R =	37.123153	deg
};
P[201]{
   GP1:
	UF : 0, UT : 1,		CONFIG : 'N U T, 0, 0, 0',
	X =	2211.963920	mm,	Y =	722.659692	mm,	Z =	973.288551	mm,
	W =	178.256690	deg,	P =	-77.272281	deg,	R =	37.387434	deg
};
P[202]{
   GP1:
	UF : 0, UT : 1,		CONFIG : 'N U T, 0, 0, 0',
	X =	2210.633943	mm,	Y =	720.017241	mm,	Z =	961.542758	mm,
	W =	114.546474	deg,	P =	-61.404714	deg,	R =	105.077214	deg
};
P[203]{
   GP1:
	UF : 0, UT : 1,		CONFIG : 'N U T, 0, 0, 0',
	X =	2199.512223	mm,	Y =	730.668272	mm,	Z =	949.262998	mm,
	W =	114.546474	deg,	P =	-61.404714	deg,	R =	105.077214	deg
};
P[204]{
   GP1:
	UF : 0, UT : 1,		CONFIG : 'N U T, 0, 0, 0',
	X =	2187.585415	mm,	Y =	740.606052	mm,	Z =	937.483291	mm,
	W =	121.150029	deg,	P =	-60.449158	deg,	R =	100.880733	deg
};
P[205]{
   GP1:
	UF : 0, UT : 1,		CONFIG : 'N U T, 0, 0, 0',
	X =	2175.033160	mm,	Y =	749.986509	mm,	Z =	925.823972	mm,
	W =	124.214455	deg,	P =	-60.286689	deg,	R =	100.179721	deg
};
P[206]{
   GP1:
	UF : 0, UT : 1,		CONFIG : 'N U T, 0, 0, 0',
	X =	2161.623114	mm,	Y =	758.613115	mm,	Z =	914.676490	mm,
	W =	130.319681	deg,	P =	-59.070939	deg,	R =	96.884778	deg
};
P[207]{
   GP1:
	UF : 0, UT : 1,		CONFIG : 'N U T, 0, 0, 0',
	X =	2147.537036	mm,	Y =	766.482149	mm,	Z =	903.724787	mm,
	W =	132.872414	deg,	P =	-59.466916	deg,	R =	97.659568	deg
};
P[208]{
   GP1:
	UF : 0, UT : 1,		CONFIG : 'N U T, 0, 0, 0',
	X =	2132.748710	mm,	Y =	773.598871	mm,	Z =	893.232764	mm,
	W =	136.300451	deg,	P =	-59.600340	deg,	R =	97.649735	deg
};
P[209]{
   GP1:
	UF : 0, UT : 1,		CONFIG : 'N U T, 0, 0, 0',
	X =	2117.370118	mm,	Y =	780.125323	mm,	Z =	883.138753	mm,
	W =	139.747908	deg,	P =	-59.223049	deg,	R =	96.714301	deg
};
P[210]{
   GP1:
	UF : 0, UT : 1,		CONFIG : 'N U T, 0, 0, 0',
	X =	2101.369960	mm,	Y =	785.654511	mm,	Z =	873.574184	mm,
	W =	143.517422	deg,	P =	-59.673233	deg,	R =	96.950304	deg
};
P[211]{
   GP1:
	UF : 0, UT : 1,		CONFIG : 'N U T, 0, 0, 0',
	X =	2084.702191	mm,	Y =	790.165598	mm,	Z =	864.680353	mm,
	W =	147.985074	deg,	P =	-59.994287	deg,	R =	96.688676	deg
};
P[212]{
   GP1:
	UF : 0, UT : 1,		CONFIG : 'N U T, 0, 0, 0',
	X =	2067.385148	mm,	Y =	793.679488	mm,	Z =	856.648599	mm,
	W =	154.035822	deg,	P =	-58.270546	deg,	R =	94.159529	deg
};
P[213]{
   GP1:
	UF : 0, UT : 1,		CONFIG : 'N U T, 0, 0, 0',
	X =	2049.601120	mm,	Y =	795.667747	mm,	Z =	849.288564	mm,
	W =	158.823567	deg,	P =	-60.828115	deg,	R =	95.341254	deg
};
P[214]{
   GP1:
	UF : 0, UT : 1,		CONFIG : 'N U T, 0, 0, 0',
	X =	2031.257564	mm,	Y =	796.583132	mm,	Z =	843.139033	mm,
	W =	165.385223	deg,	P =	-58.763294	deg,	R =	92.847131	deg
};
P[215]{
   GP1:
	UF : 0, UT : 1,		CONFIG : 'N U T, 0, 0, 0',
	X =	2012.669205	mm,	Y =	795.865812	mm,	Z =	837.984982	mm,
	W =	172.315708	deg,	P =	-59.503915	deg,	R =	91.752337	deg
};
P[216]{
   GP1:
	UF : 0, UT : 1,		CONFIG : 'N U T, 0, 0, 0',
	X =	1993.854802	mm,	Y =	793.803678	mm,	Z =	834.083937	mm,
	W =	178.933403	deg,	P =	-58.248343	deg,	R =	90.119432	deg
};
P[217]{
   GP1:
	UF : 0, UT : 1,		CONFIG : 'N U T, 0, 0, 0',
	X =	1975.037516	mm,	Y =	790.342207	mm,	Z =	831.322541	mm,
	W =	-174.706084	deg,	P =	-57.284930	deg,	R =	88.789544	deg
};
P[218]{
   GP1:
	UF : 0, UT : 1,		CONFIG : 'N U T, 0, 0, 0',
	X =	1956.446874	mm,	Y =	785.370491	mm,	Z =	829.689682	mm,
	W =	-166.914980	deg,	P =	-58.308430	deg,	R =	86.717255	deg
};
P[219]{
   GP1:
	UF : 0, UT : 1,		CONFIG : 'N U T, 0, 0, 0',
	X =	1938.186722	mm,	Y =	779.073212	mm,	Z =	829.424816	mm,
	W =	-159.832035	deg,	P =	-57.573918	deg,	R =	84.987847	deg
};
P[220]{
   GP1:
	UF : 0, UT : 1,		CONFIG : 'N U T, 0, 0, 0',
	X =	1920.306939	mm,	Y =	771.654234	mm,	Z =	830.278063	mm,
	W =	-154.377165	deg,	P =	-56.365933	deg,	R =	84.001109	deg
};
P[221]{
   GP1:
	UF : 0, UT : 1,		CONFIG : 'N U T, 0, 0, 0',
	X =	1903.004185	mm,	Y =	763.153813	mm,	Z =	832.223725	mm,
	W =	-149.185346	deg,	P =	-54.992711	deg,	R =	83.329853	deg
};
P[222]{
   GP1:
	UF : 0, UT : 1,		CONFIG : 'N U T, 0, 0, 0',
	X =	1886.347586	mm,	Y =	753.633586	mm,	Z =	835.086604	mm,
	W =	-143.002359	deg,	P =	-54.825477	deg,	R =	81.470156	deg
};
P[223]{
   GP1:
	UF : 0, UT : 1,		CONFIG : 'N U T, 0, 0, 0',
	X =	1870.205911	mm,	Y =	743.412698	mm,	Z =	838.814012	mm,
	W =	-139.245254	deg,	P =	-53.831117	deg,	R =	81.041948	deg
};
P[224]{
   GP1:
	UF : 0, UT : 1,		CONFIG : 'N U T, 0, 0, 0',
	X =	1854.765527	mm,	Y =	732.489711	mm,	Z =	843.357765	mm,
	W =	-135.572909	deg,	P =	-52.621104	deg,	R =	80.917510	deg
};
P[225]{
   GP1:
	UF : 0, UT : 1,		CONFIG : 'N U T, 0, 0, 0',
	X =	1839.918740	mm,	Y =	720.953350	mm,	Z =	848.513639	mm,
	W =	-131.577952	deg,	P =	-52.195149	deg,	R =	79.869871	deg
};
P[226]{
   GP1:
	UF : 0, UT : 1,		CONFIG : 'N U T, 0, 0, 0',
	X =	1825.638075	mm,	Y =	708.977521	mm,	Z =	854.323456	mm,
	W =	-129.431752	deg,	P =	-51.041080	deg,	R =	80.369176	deg
};
P[227]{
   GP1:
	UF : 0, UT : 1,		CONFIG : 'N U T, 0, 0, 0',
	X =	1812.165672	mm,	Y =	696.456489	mm,	Z =	860.739368	mm,
	W =	-125.551838	deg,	P =	-50.307441	deg,	R =	79.707313	deg
};
P[228]{
   GP1:
	UF : 0, UT : 1,		CONFIG : 'N U T, 0, 0, 0',
	X =	1799.174772	mm,	Y =	683.573230	mm,	Z =	867.653466	mm,
	W =	-123.393599	deg,	P =	-49.614677	deg,	R =	79.708101	deg
};
P[229]{
   GP1:
	UF : 0, UT : 1,		CONFIG : 'N U T, 0, 0, 0',
	X =	1786.680255	mm,	Y =	670.394968	mm,	Z =	874.953431	mm,
	W =	-121.319993	deg,	P =	-49.053307	deg,	R =	79.576233	deg
};
P[230]{
   GP1:
	UF : 0, UT : 1,		CONFIG : 'N U T, 0, 0, 0',
	X =	1788.790373	mm,	Y =	667.087702	mm,	Z =	865.042298	mm,
	W =	-112.894717	deg,	P =	-25.103856	deg,	R =	65.586792	deg
};
P[231]{
   GP1:
	UF : 0, UT : 1,		CONFIG : 'N U T, 0, 0, 0',
	X =	1795.110314	mm,	Y =	673.784975	mm,	Z =	861.313059	mm,
	W =	-112.894717	deg,	P =	-25.103856	deg,	R =	65.586792	deg
};
P[232]{
   GP1:
	UF : 0, UT : 1,		CONFIG : 'N U T, 0, 0, 0',
	X =	1808.030100	mm,	Y =	686.942442	mm,	Z =	854.154919	mm,
	W =	-113.782437	deg,	P =	-25.665192	deg,	R =	65.043035	deg
};
P[233]{
   GP1:
	UF : 0, UT : 1,		CONFIG : 'N U T, 0, 0, 0',
	X =	1821.600888	mm,	Y =	699.569445	mm,	Z =	847.579934	mm,
	W =	-114.891470	deg,	P =	-27.216727	deg,	R =	63.166821	deg
};
P[234]{
   GP1:
	UF : 0, UT : 1,		CONFIG : 'N U T, 0, 0, 0',
	X =	1835.742983	mm,	Y =	711.902097	mm,	Z =	841.550711	mm,
	W =	-117.070096	deg,	P =	-28.041667	deg,	R =	62.714169	deg
};
P[235]{
   GP1:
	UF : 0, UT : 1,		CONFIG : 'N U T, 0, 0, 0',
	X =	1850.533198	mm,	Y =	723.656244	mm,	Z =	836.115561	mm,
	W =	-118.661199	deg,	P =	-29.561060	deg,	R =	61.174618	deg
};
P[236]{
   GP1:
	UF : 0, UT : 1,		CONFIG : 'N U T, 0, 0, 0',
	X =	1865.940953	mm,	Y =	734.911638	mm,	Z =	831.364188	mm,
	W =	-121.090778	deg,	P =	-30.729421	deg,	R =	60.378883	deg
};
P[237]{
   GP1:
	UF : 0, UT : 1,		CONFIG : 'N U T, 0, 0, 0',
	X =	1881.982822	mm,	Y =	745.486458	mm,	Z =	827.328502	mm,
	W =	-123.211324	deg,	P =	-32.325765	deg,	R =	59.006417	deg
};
P[238]{
   GP1:
	UF : 0, UT : 1,		CONFIG : 'N U T, 0, 0, 0',
	X =	1898.731676	mm,	Y =	755.104300	mm,	Z =	824.176223	mm,
	W =	-124.222004	deg,	P =	-35.079399	deg,	R =	56.109562	deg
};
P[239]{
   GP1:
	UF : 0, UT : 1,		CONFIG : 'N U T, 0, 0, 0',
	X =	1916.064445	mm,	Y =	764.010533	mm,	Z =	822.041665	mm,
	W =	-127.844015	deg,	P =	-36.423755	deg,	R =	55.559156	deg
};
P[240]{
   GP1:
	UF : 0, UT : 1,		CONFIG : 'N U T, 0, 0, 0',
	X =	1933.944601	mm,	Y =	771.816419	mm,	Z =	820.957051	mm,
	W =	-131.433696	deg,	P =	-38.413024	deg,	R =	54.305929	deg
};
P[241]{
   GP1:
	UF : 0, UT : 1,		CONFIG : 'N U T, 0, 0, 0',
	X =	1952.307562	mm,	Y =	778.412634	mm,	Z =	821.023896	mm,
	W =	-135.083228	deg,	P =	-40.657714	deg,	R =	52.852116	deg
};
P[242]{
   GP1:
	UF : 0, UT : 1,		CONFIG : 'N U T, 0, 0, 0',
	X =	1971.047050	mm,	Y =	783.804938	mm,	Z =	822.125524	mm,
	W =	-137.516092	deg,	P =	-43.308865	deg,	R =	50.874971	deg
};
P[243]{
   GP1:
	UF : 0, UT : 1,		CONFIG : 'N U T, 0, 0, 0',
	X =	1989.947977	mm,	Y =	787.715719	mm,	Z =	824.586249	mm,
	W =	-141.244484	deg,	P =	-46.199024	deg,	R =	49.034418	deg
};
P[244]{
   GP1:
	UF : 0, UT : 1,		CONFIG : 'N U T, 0, 0, 0',
	X =	2008.910510	mm,	Y =	790.225958	mm,	Z =	828.290791	mm,
	W =	-145.399704	deg,	P =	-48.570530	deg,	R =	47.767561	deg
};
P[245]{
   GP1:
	UF : 0, UT : 1,		CONFIG : 'N U T, 0, 0, 0',
	X =	2027.720252	mm,	Y =	791.219720	mm,	Z =	833.202874	mm,
	W =	-149.412709	deg,	P =	-51.212073	deg,	R =	46.311919	deg
};
P[246]{
   GP1:
	UF : 0, UT : 1,		CONFIG : 'N U T, 0, 0, 0',
	X =	2046.198194	mm,	Y =	790.660430	mm,	Z =	839.280866	mm,
	W =	-153.005716	deg,	P =	-54.203892	deg,	R =	44.630375	deg
};
P[247]{
   GP1:
	UF : 0, UT : 1,		CONFIG : 'N U T, 0, 0, 0',
	X =	2064.279711	mm,	Y =	788.757896	mm,	Z =	846.359062	mm,
	W =	-156.161022	deg,	P =	-56.847031	deg,	R =	43.231228	deg
};
P[248]{
   GP1:
	UF : 0, UT : 1,		CONFIG : 'N U T, 0, 0, 0',
	X =	2081.929608	mm,	Y =	785.686889	mm,	Z =	854.214817	mm,
	W =	-158.092117	deg,	P =	-59.623063	deg,	R =	41.707721	deg
};
P[249]{
   GP1:
	UF : 0, UT : 1,		CONFIG : 'N U T, 0, 0, 0',
	X =	2098.746648	mm,	Y =	781.356725	mm,	Z =	863.089635	mm,
	W =	-163.019127	deg,	P =	-61.358368	deg,	R =	41.166186	deg
};
P[250]{
   GP1:
	UF : 0, UT : 1,		CONFIG : 'N U T, 0, 0, 0',
	X =	2115.001897	mm,	Y =	775.930656	mm,	Z =	872.573689	mm,
	W =	-165.694633	deg,	P =	-63.454180	deg,	R =	40.250102	deg
};
P[251]{
   GP1:
	UF : 0, UT : 1,		CONFIG : 'N U T, 0, 0, 0',
	X =	2130.637611	mm,	Y =	769.656331	mm,	Z =	882.630893	mm,
	W =	-168.603879	deg,	P =	-64.838353	deg,	R =	39.727151	deg
};
P[252]{
   GP1:
	UF : 0, UT : 1,		CONFIG : 'N U T, 0, 0, 0',
	X =	2145.543105	mm,	Y =	762.462775	mm,	Z =	893.151275	mm,
	W =	-170.723537	deg,	P =	-67.069867	deg,	R =	38.859537	deg
};
P[253]{
   GP1:
	UF : 0, UT : 1,		CONFIG : 'N U T, 0, 0, 0',
	X =	2159.970027	mm,	Y =	754.698939	mm,	Z =	904.085135	mm,
	W =	-172.973150	deg,	P =	-67.910942	deg,	R =	38.578655	deg
};
P[254]{
   GP1:
	UF : 0, UT : 1,		CONFIG : 'N U T, 0, 0, 0',
	X =	2173.638918	mm,	Y =	746.200012	mm,	Z =	915.349357	mm,
	W =	-175.114782	deg,	P =	-69.705791	deg,	R =	38.010678	deg
};
P[255]{
   GP1:
	UF : 0, UT : 1,		CONFIG : 'N U T, 0, 0, 0',
	X =	2186.630270	mm,	Y =	736.996558	mm,	Z =	926.889461	mm,
	W =	-176.258303	deg,	P =	-72.272001	deg,	R =	37.414080	deg
};
P[256]{
   GP1:
	UF : 0, UT : 1,		CONFIG : 'N U T, 0, 0, 0',
	X =	2198.700650	mm,	Y =	727.329744	mm,	Z =	938.662294	mm,
	W =	-178.629432	deg,	P =	-73.892429	deg,	R =	37.209468	deg
};
P[257]{
   GP1:
	UF : 0, UT : 1,		CONFIG : 'N U T, 0, 0, 0',
	X =	2204.675255	mm,	Y =	722.089951	mm,	Z =	944.753916	mm,
	W =	-179.430188	deg,	P =	-75.982868	deg,	R =	37.153060	deg
};
P[258]{
   GP1:
	UF : 0, UT : 1,		CONFIG : 'N U T, 0, 0, 0',
	X =	2203.816969	mm,	Y =	718.792006	mm,	Z =	934.134933	mm,
	W =	125.563407	deg,	P =	-58.832419	deg,	R =	96.043345	deg
};
P[259]{
   GP1:
	UF : 0, UT : 1,		CONFIG : 'N U T, 0, 0, 0',
	X =	2191.489246	mm,	Y =	728.648930	mm,	Z =	922.160397	mm,
	W =	125.563407	deg,	P =	-58.832419	deg,	R =	96.043345	deg
};
P[260]{
   GP1:
	UF : 0, UT : 1,		CONFIG : 'N U T, 0, 0, 0',
	X =	2178.667652	mm,	Y =	737.907736	mm,	Z =	910.503493	mm,
	W =	128.108485	deg,	P =	-58.686962	deg,	R =	95.872655	deg
};
P[261]{
   GP1:
	UF : 0, UT : 1,		CONFIG : 'N U T, 0, 0, 0',
	X =	2165.172132	mm,	Y =	746.507213	mm,	Z =	899.171743	mm,
	W =	131.039613	deg,	P =	-58.646363	deg,	R =	95.930261	deg
};
P[262]{
   GP1:
	UF : 0, UT : 1,		CONFIG : 'N U T, 0, 0, 0',
	X =	2151.084713	mm,	Y =	754.541657	mm,	Z =	888.097364	mm,
	W =	133.113416	deg,	P =	-58.977408	deg,	R =	96.652456	deg
};
P[263]{
   GP1:
	UF : 0, UT : 1,		CONFIG : 'N U T, 0, 0, 0',
	X =	2136.406182	mm,	Y =	762.019885	mm,	Z =	877.426014	mm,
	W =	136.498194	deg,	P =	-58.491446	deg,	R =	95.661981	deg
};
P[264]{
   GP1:
	UF : 0, UT : 1,		CONFIG : 'N U T, 0, 0, 0',
	X =	2121.006496	mm,	Y =	768.479866	mm,	Z =	867.285140	mm,
	W =	140.509067	deg,	P =	-58.623652	deg,	R =	95.736227	deg
};
P[265]{
   GP1:
	UF : 0, UT : 1,		CONFIG : 'N U T, 0, 0, 0',
	X =	2104.980332	mm,	Y =	774.180374	mm,	Z =	857.565587	mm,
	W =	143.412346	deg,	P =	-59.167821	deg,	R =	96.283754	deg
};
P[266]{
   GP1:
	UF : 0, UT : 1,		CONFIG : 'N U T, 0, 0, 0',
	X =	2088.296872	mm,	Y =	778.889366	mm,	Z =	848.588833	mm,
	W =	148.376393	deg,	P =	-58.681869	deg,	R =	95.174632	deg
};
P[267]{
   GP1:
	UF : 0, UT : 1,		CONFIG : 'N U T, 0, 0, 0',
	X =	2070.988163	mm,	Y =	782.444746	mm,	Z =	840.330727	mm,
	W =	153.333375	deg,	P =	-58.683508	deg,	R =	94.606914	deg
};
P[268]{
   GP1:
	UF : 0, UT : 1,		CONFIG : 'N U T, 0, 0, 0',
	X =	2053.108276	mm,	Y =	784.703394	mm,	Z =	832.970677	mm,
	W =	158.970248	deg,	P =	-58.784135	deg,	R =	93.903386	deg
};
P[269]{
   GP1:
	UF : 0, UT : 1,		CONFIG : 'N U T, 0, 0, 0',
	X =	2034.738769	mm,	Y =	785.728174	mm,	Z =	826.616851	mm,
	W =	164.929815	deg,	P =	-57.710494	deg,	R =	92.419263	deg
};
P[270]{
   GP1:
	UF : 0, UT : 1,		CONFIG : 'N U T, 0, 0, 0',
	X =	2016.069370	mm,	Y =	785.214827	mm,	Z =	821.272149	mm,
	W =	171.355795	deg,	P =	-58.420680	deg,	R =	91.645849	deg
};
P[271]{
   GP1:
	UF : 0, UT : 1,		CONFIG : 'N U T, 0, 0, 0',
	X =	1997.186019	mm,	Y =	783.233968	mm,	Z =	817.300828	mm,
	W =	178.274728	deg,	P =	-56.867593	deg,	R =	90.130792	deg
};
P[272]{
   GP1:
	UF : 0, UT : 1,		CONFIG : 'N U T, 0, 0, 0',
	X =	1978.295545	mm,	Y =	779.768732	mm,	Z =	814.385416	mm,
	W =	-175.018868	deg,	P =	-57.312842	deg,	R =	88.853188	deg
};
P[273]{
   GP1:
	UF : 0, UT : 1,		CONFIG : 'N U T, 0, 0, 0',
	X =	1959.506397	mm,	Y =	775.038723	mm,	Z =	812.646176	mm,
	W =	-168.853198	deg,	P =	-56.881693	deg,	R =	87.568198	deg
};
P[274]{
   GP1:
	UF : 0, UT : 1,		CONFIG : 'N U T, 0, 0, 0',
	X =	1941.124708	mm,	Y =	768.852803	mm,	Z =	812.223891	mm,
	W =	-161.568179	deg,	P =	-56.425234	deg,	R =	85.954363	deg
};
P[275]{
   GP1:
	UF : 0, UT : 1,		CONFIG : 'N U T, 0, 0, 0',
	X =	1923.128511	mm,	Y =	761.479043	mm,	Z =	812.945834	mm,
	W =	-155.519022	deg,	P =	-55.782937	deg,	R =	84.657473	deg
};
P[276]{
   GP1:
	UF : 0, UT : 1,		CONFIG : 'N U T, 0, 0, 0',
	X =	1905.600474	mm,	Y =	753.105439	mm,	Z =	814.699788	mm,
	W =	-150.633834	deg,	P =	-54.729188	deg,	R =	83.934569	deg
};
P[277]{
   GP1:
	UF : 0, UT : 1,		CONFIG : 'N U T, 0, 0, 0',
	X =	1888.781048	mm,	Y =	743.704193	mm,	Z =	817.542758	mm,
	W =	-145.592142	deg,	P =	-53.391735	deg,	R =	83.466867	deg
};
P[278]{
   GP1:
	UF : 0, UT : 1,		CONFIG : 'N U T, 0, 0, 0',
	X =	1872.450700	mm,	Y =	733.541240	mm,	Z =	821.151826	mm,
	W =	-141.814763	deg,	P =	-52.602796	deg,	R =	83.009263	deg
};
P[279]{
   GP1:
	UF : 0, UT : 1,		CONFIG : 'N U T, 0, 0, 0',
	X =	1856.815478	mm,	Y =	722.618997	mm,	Z =	825.479566	mm,
	W =	-136.371119	deg,	P =	-52.713559	deg,	R =	81.109542	deg
};
P[280]{
   GP1:
	UF : 0, UT : 1,		CONFIG : 'N U T, 0, 0, 0',
	X =	1841.827580	mm,	Y =	711.176791	mm,	Z =	830.742454	mm,
	W =	-134.848916	deg,	P =	-50.517619	deg,	R =	82.894751	deg
};
P[281]{
   GP1:
	UF : 0, UT : 1,		CONFIG : 'N U T, 0, 0, 0',
	X =	1827.477143	mm,	Y =	699.113263	mm,	Z =	836.482231	mm,
	W =	-130.995613	deg,	P =	-50.234184	deg,	R =	81.914739	deg
};
P[282]{
   GP1:
	UF : 0, UT : 1,		CONFIG : 'N U T, 0, 0, 0',
	X =	1813.773330	mm,	Y =	686.603834	mm,	Z =	842.841244	mm,
	W =	-127.891557	deg,	P =	-49.582988	deg,	R =	81.577089	deg
};
P[283]{
   GP1:
	UF : 0, UT : 1,		CONFIG : 'N U T, 0, 0, 0',
	X =	1800.645940	mm,	Y =	673.767647	mm,	Z =	849.616779	mm,
	W =	-124.964724	deg,	P =	-49.282700	deg,	R =	80.824111	deg
};
P[284]{
   GP1:
	UF : 0, UT : 1,		CONFIG : 'N U T, 0, 0, 0',
	X =	1794.233203	mm,	Y =	667.178191	mm,	Z =	853.224570	mm,
	W =	-123.385439	deg,	P =	-48.746709	deg,	R =	80.911243	deg
};
P[285]{
   GP1:
	UF : 0, UT : 1,		CONFIG : 'N U T, 0, 0, 0',
	X =	1799.738008	mm,	Y =	667.023672	mm,	Z =	841.741746	mm,
	W =	-115.995568	deg,	P =	-25.767244	deg,	R =	65.580745	deg
};
P[286]{
   GP1:
	UF : 0, UT : 1,		CONFIG : 'N U T, 0, 0, 0',
	X =	1812.972900	mm,	Y =	679.978518	mm,	Z =	834.830931	mm,
	W =	-115.995568	deg,	P =	-25.767244	deg,	R =	65.580745	deg
};
P[287]{
   GP1:
	UF : 0, UT : 1,		CONFIG : 'N U T, 0, 0, 0',
	X =	1826.627340	mm,	Y =	692.514581	mm,	Z =	828.402483	mm,
	W =	-117.194432	deg,	P =	-26.763598	deg,	R =	64.508843	deg
};
P[288]{
   GP1:
	UF : 0, UT : 1,		CONFIG : 'N U T, 0, 0, 0',
	X =	1840.943248	mm,	Y =	704.533094	mm,	Z =	822.664025	mm,
	W =	-119.504668	deg,	P =	-28.008724	deg,	R =	63.441334	deg
};
P[289]{
   GP1:
	UF : 0, UT : 1,		CONFIG : 'N U T, 0, 0, 0',
	X =	1855.901804	mm,	Y =	716.035261	mm,	Z =	817.498263	mm,
	W =	-121.131061	deg,	P =	-29.415055	deg,	R =	62.034792	deg
};
P[290]{
   GP1:
	UF : 0, UT : 1,		CONFIG : 'N U T, 0, 0, 0',
	X =	1871.448313	mm,	Y =	727.006331	mm,	Z =	812.946951	mm,
	W =	-122.639009	deg,	P =	-30.875486	deg,	R =	60.598295	deg
};
P[291]{
   GP1:
	UF : 0, UT : 1,		CONFIG : 'N U T, 0, 0, 0',
	X =	1887.644942	mm,	Y =	737.239384	mm,	Z =	809.313299	mm,
	W =	-125.762195	deg,	P =	-32.353097	deg,	R =	59.576677	deg
};
P[292]{
   GP1:
	UF : 0, UT : 1,		CONFIG : 'N U T, 0, 0, 0',
	X =	1904.455478	mm,	Y =	746.718380	mm,	Z =	806.390842	mm,
	W =	-127.525795	deg,	P =	-34.216548	deg,	R =	57.867830	deg
};
P[293]{
   GP1:
	UF : 0, UT : 1,		CONFIG : 'N U T, 0, 0, 0',
	X =	1921.840467	mm,	Y =	755.261188	mm,	Z =	804.499232	mm,
	W =	-130.496498	deg,	P =	-36.164956	deg,	R =	56.401992	deg
};
P[294]{
   GP1:
	UF : 0, UT : 1,		CONFIG : 'N U T, 0, 0, 0',
	X =	1939.778378	mm,	Y =	762.681190	mm,	Z =	803.666177	mm,
	W =	-133.090688	deg,	P =	-38.672371	deg,	R =	54.379866	deg
};
P[295]{
   GP1:
	UF : 0, UT : 1,		CONFIG : 'N U T, 0, 0, 0',
	X =	1958.156223	mm,	Y =	768.982875	mm,	Z =	803.955958	mm,
	W =	-136.268957	deg,	P =	-40.922057	deg,	R =	52.819448	deg
};
P[296]{
   GP1:
	UF : 0, UT : 1,		CONFIG : 'N U T, 0, 0, 0',
	X =	1976.807219	mm,	Y =	773.937463	mm,	Z =	805.626908	mm,
	W =	-141.819718	deg,	P =	-42.596621	deg,	R =	52.158934	deg
};
P[297]{
   GP1:
	UF : 0, UT : 1,		CONFIG : 'N U T, 0, 0, 0',
	X =	1995.667615	mm,	Y =	777.405349	mm,	Z =	808.391408	mm,
	W =	-144.744826	deg,	P =	-45.600989	deg,	R =	50.033966	deg
};
P[298]{
   GP1:
	UF : 0, UT : 1,		CONFIG : 'N U T, 0, 0, 0',
	X =	2014.541737	mm,	Y =	779.523109	mm,	Z =	812.323714	mm,
	W =	-147.879018	deg,	P =	-48.304042	deg,	R =	48.291914	deg
};
P[299]{
   GP1:
	UF : 0, UT : 1,		CONFIG : 'N U T, 0, 0, 0',
	X =	2033.154870	mm,	Y =	780.068063	mm,	Z =	817.549344	mm,
	W =	-151.977006	deg,	P =	-51.134349	deg,	R =	46.647644	deg
};
P[300]{
   GP1:
	UF : 0, UT : 1,		CONFIG : 'N U T, 0, 0, 0',
	X =	2051.569828	mm,	Y =	779.273428	mm,	Z =	823.670723	mm,
	W =	-153.500855	deg,	P =	-54.529320	deg,	R =	44.465612	deg
};
P[301]{
   GP1:
	UF : 0, UT : 1,		CONFIG : 'N U T, 0, 0, 0',
	X =	2069.466226	mm,	Y =	777.359631	mm,	Z =	830.968225	mm,
	W =	-159.593928	deg,	P =	-55.031082	deg,	R =	44.600885	deg
};
P[302]{
   GP1:
	UF : 0, UT : 1,		CONFIG : 'N U T, 0, 0, 0',
	X =	2086.743701	mm,	Y =	773.827276	mm,	Z =	839.005009	mm,
	W =	-161.092583	deg,	P =	-59.253834	deg,	R =	42.204463	deg
};
P[303]{
   GP1:
	UF : 0, UT : 1,		CONFIG : 'N U T, 0, 0, 0',
	X =	2103.489910	mm,	Y =	769.343597	mm,	Z =	847.893013	mm,
	W =	-164.251493	deg,	P =	-60.952268	deg,	R =	41.450469	deg
};
P[304]{
   GP1:
	UF : 0, UT : 1,		CONFIG : 'N U T, 0, 0, 0',
	X =	2119.576979	mm,	Y =	763.924499	mm,	Z =	857.466693	mm,
	W =	-168.321827	deg,	P =	-61.784614	deg,	R =	41.097149	deg
};
P[305]{
   GP1:
	UF : 0, UT : 1,		CONFIG : 'N U T, 0, 0, 0',
	X =	2134.980205	mm,	Y =	757.453412	mm,	Z =	867.510721	mm,
	W =	-170.280103	deg,	P =	-64.295401	deg,	R =	39.968842	deg
};
P[306]{
   GP1:
	UF : 0, UT : 1,		CONFIG : 'N U T, 0, 0, 0',
	X =	2149.802935	mm,	Y =	750.223076	mm,	Z =	878.009869	mm,
	W =	-171.800351	deg,	P =	-66.388167	deg,	R =	39.126956	deg
};
P[307]{
   GP1:
	UF : 0, UT : 1,		CONFIG : 'N U T, 0, 0, 0',
	X =	2163.821057	mm,	Y =	742.228565	mm,	Z =	888.991939	mm,
	W =	-174.391635	deg,	P =	-68.083527	deg,	R =	38.493391	deg
};
P[308]{
   GP1:
	UF : 0, UT : 1,		CONFIG : 'N U T, 0, 0, 0',
	X =	2177.402549	mm,	Y =	733.700255	mm,	Z =	900.282174	mm,
	W =	-176.152104	deg,	P =	-69.019652	deg,	R =	38.145690	deg
};
P[309]{
   GP1:
	UF : 0, UT : 1,		CONFIG : 'N U T, 0, 0, 0',
	X =	2190.346577	mm,	Y =	724.614826	mm,	Z =	911.845459	mm,
	W =	-178.120189	deg,	P =	-70.233012	deg,	R =	37.729539	deg
};
P[310]{
   GP1:
	UF : 0, UT : 1,		CONFIG : 'N U T, 0, 0, 0',
	X =	2202.694936	mm,	Y =	714.914755	mm,	Z =	923.556653	mm,
	W =	-178.703860	deg,	P =	-72.952637	deg,	R =	37.297311	deg
};
P[311]{
   GP1:
	UF : 0, UT : 1,		CONFIG : 'N U T, 0, 0, 0',
	X =	2201.404636	mm,	Y =	711.028462	mm,	Z =	913.191908	mm,
	W =	127.515480	deg,	P =	-58.303664	deg,	R =	94.795282	deg
};
P[312]{
   GP1:
	UF : 0, UT : 1,		CONFIG : 'N U T, 0, 0, 0',
	X =	2188.847427	mm,	Y =	720.632845	mm,	Z =	901.360691	mm,
	W =	127.515480	deg,	P =	-58.303664	deg,	R =	94.795282	deg
};
P[313]{
   GP1:
	UF : 0, UT : 1,		CONFIG : 'N U T, 0, 0, 0',
	X =	2175.775467	mm,	Y =	729.613403	mm,	Z =	889.885403	mm,
	W =	130.431489	deg,	P =	-57.956204	deg,	R =	94.281537	deg
};
P[314]{
   GP1:
	UF : 0, UT : 1,		CONFIG : 'N U T, 0, 0, 0',
	X =	2162.196014	mm,	Y =	738.125623	mm,	Z =	878.599793	mm,
	W =	132.309880	deg,	P =	-58.039511	deg,	R =	94.652360	deg
};
P[315]{
   GP1:
	UF : 0, UT : 1,		CONFIG : 'N U T, 0, 0, 0',
	X =	2147.952894	mm,	Y =	745.882892	mm,	Z =	867.723284	mm,
	W =	135.282558	deg,	P =	-58.157044	deg,	R =	95.037151	deg
};
P[316]{
   GP1:
	UF : 0, UT : 1,		CONFIG : 'N U T, 0, 0, 0',
	X =	2133.074779	mm,	Y =	753.033887	mm,	Z =	857.248499	mm,
	W =	138.642631	deg,	P =	-57.730968	deg,	R =	94.349171	deg
};
P[317]{
   GP1:
	UF : 0, UT : 1,		CONFIG : 'N U T, 0, 0, 0',
	X =	2117.505353	mm,	Y =	759.309365	mm,	Z =	847.344219	mm,
	W =	143.246634	deg,	P =	-56.779853	deg,	R =	93.017799	deg
};
P[318]{
   GP1:
	UF : 0, UT : 1,		CONFIG : 'N U T, 0, 0, 0',
	X =	2101.281726	mm,	Y =	764.560706	mm,	Z =	837.931690	mm,
	W =	146.813060	deg,	P =	-57.235948	deg,	R =	93.615317	deg
};
P[319]{
   GP1:
	UF : 0, UT : 1,		CONFIG : 'N U T, 0, 0, 0',
	X =	2084.463977	mm,	Y =	768.971488	mm,	Z =	829.092533	mm,
	W =	150.371827	deg,	P =	-57.415808	deg,	R =	93.667594	deg
};
P[320]{
   GP1:
	UF : 0, UT : 1,		CONFIG : 'N U T, 0, 0, 0',
	X =	2066.996304	mm,	Y =	772.028240	mm,	Z =	821.293970	mm,
	W =	156.629380	deg,	P =	-56.338941	deg,	R =	92.378879	deg
};
P[321]{
   GP1:
	UF : 0, UT : 1,		CONFIG : 'N U T, 0, 0, 0',
	X =	2048.992226	mm,	Y =	773.834665	mm,	Z =	814.241198	mm,
	W =	161.489939	deg,	P =	-56.762026	deg,	R =	92.313692	deg
};
P[322]{
   GP1:
	UF : 0, UT : 1,		CONFIG : 'N U T, 0, 0, 0',
	X =	2030.557173	mm,	Y =	774.531371	mm,	Z =	808.143316	mm,
	W =	166.622760	deg,	P =	-55.695587	deg,	R =	91.333780	deg
};
P[323]{
   GP1:
	UF : 0, UT : 1,		CONFIG : 'N U T, 0, 0, 0',
	X =	2011.899502	mm,	Y =	773.666167	mm,	Z =	803.057684	mm,
	W =	172.825667	deg,	P =	-56.763385	deg,	R =	90.969871	deg
};
P[324]{
   GP1:
	UF : 0, UT : 1,		CONFIG : 'N U T, 0, 0, 0',
	X =	1993.096991	mm,	Y =	771.222223	mm,	Z =	799.433604	mm,
	W =	-179.948006	deg,	P =	-55.769425	deg,	R =	89.781042	deg
};
P[325]{
   GP1:
	UF : 0, UT : 1,		CONFIG : 'N U T, 0, 0, 0',
	X =	1974.242888	mm,	Y =	767.472073	mm,	Z =	796.886042	mm,
	W =	-174.267904	deg,	P =	-55.058388	deg,	R =	88.938874	deg
};
P[326]{
   GP1:
	UF : 0, UT : 1,		CONFIG : 'N U T, 0, 0, 0',
	X =	1955.655106	mm,	Y =	762.276160	mm,	Z =	795.611168	mm,
	W =	-167.789443	deg,	P =	-54.345075	deg,	R =	88.006970	deg
};
P[327]{
   GP1:
	UF : 0, UT : 1,		CONFIG : 'N U T, 0, 0, 0',
	X =	1937.389464	mm,	Y =	755.791314	mm,	Z =	795.448093	mm,
	W =	-161.500637	deg,	P =	-54.380471	deg,	R =	86.794506	deg
};
P[328]{
   GP1:
	UF : 0, UT : 1,		CONFIG : 'N U T, 0, 0, 0',
	X =	1919.529984	mm,	Y =	748.206075	mm,	Z =	796.317711	mm,
	W =	-155.490726	deg,	P =	-54.568852	deg,	R =	85.328035	deg
};
P[329]{
   GP1:
	UF : 0, UT : 1,		CONFIG : 'N U T, 0, 0, 0',
	X =	1902.298878	mm,	Y =	739.539127	mm,	Z =	798.375943	mm,
	W =	-149.790205	deg,	P =	-53.659367	deg,	R =	84.436038	deg
};
P[330]{
   GP1:
	UF : 0, UT : 1,		CONFIG : 'N U T, 0, 0, 0',
	X =	1885.527535	mm,	Y =	730.066456	mm,	Z =	801.328723	mm,
	W =	-146.278335	deg,	P =	-52.349456	deg,	R =	84.485529	deg
};
P[331]{
   GP1:
	UF : 0, UT : 1,		CONFIG : 'N U T, 0, 0, 0',
	X =	1869.472475	mm,	Y =	719.723912	mm,	Z =	805.083658	mm,
	W =	-141.021984	deg,	P =	-52.150974	deg,	R =	83.177645	deg
};
P[332]{
   GP1:
	UF : 0, UT : 1,		CONFIG : 'N U T, 0, 0, 0',
	X =	1854.083836	mm,	Y =	708.718330	mm,	Z =	809.758473	mm,
	W =	-137.916041	deg,	P =	-50.658840	deg,	R =	83.689112	deg
};
P[333]{
   GP1:
	UF : 0, UT : 1,		CONFIG : 'N U T, 0, 0, 0',
	X =	1839.244572	mm,	Y =	697.121222	mm,	Z =	814.991178	mm,
	W =	-134.531480	deg,	P =	-50.233803	deg,	R =	83.102984	deg
};
P[334]{
   GP1:
	UF : 0, UT : 1,		CONFIG : 'N U T, 0, 0, 0',
	X =	1825.071799	mm,	Y =	685.031927	mm,	Z =	820.880107	mm,
	W =	-131.530972	deg,	P =	-49.417357	deg,	R =	83.064333	deg
};
P[335]{
   GP1:
	UF : 0, UT : 1,		CONFIG : 'N U T, 0, 0, 0',
	X =	1811.391975	mm,	Y =	672.534906	mm,	Z =	827.234608	mm,
	W =	-128.954916	deg,	P =	-48.982857	deg,	R =	82.722138	deg
};
P[336]{
   GP1:
	UF : 0, UT : 1,		CONFIG : 'N U T, 0, 0, 0',
	X =	1798.422717	mm,	Y =	659.655723	mm,	Z =	834.177838	mm,
	W =	-126.557171	deg,	P =	-48.011920	deg,	R =	83.143825	deg
};
P[337]{
   GP1:
	UF : 0, UT : 1,		CONFIG : 'N U T, 0, 0, 0',
	X =	1799.343934	mm,	Y =	654.469331	mm,	Z =	825.442095	mm,
	W =	-116.493835	deg,	P =	-25.270459	deg,	R =	66.442325	deg
};
P[338]{
   GP1:
	UF : 0, UT : 1,		CONFIG : 'N U T, 0, 0, 0',
	X =	1805.908173	mm,	Y =	660.989860	mm,	Z =	821.934540	mm,
	W =	-116.493835	deg,	P =	-25.270459	deg,	R =	66.442325	deg
};
P[339]{
   GP1:
	UF : 0, UT : 1,		CONFIG : 'N U T, 0, 0, 0',
	X =	1812.656403	mm,	Y =	667.562771	mm,	Z =	818.473402	mm,
	W =	-117.262403	deg,	P =	-25.474793	deg,	R =	66.351870	deg
};
P[340]{
   GP1:
	UF : 0, UT : 1,		CONFIG : 'N U T, 0, 0, 0',
	X =	1826.524041	mm,	Y =	680.200349	mm,	Z =	812.058063	mm,
	W =	-118.862456	deg,	P =	-26.340250	deg,	R =	65.538213	deg
};
P[341]{
   GP1:
	UF : 0, UT : 1,		CONFIG : 'N U T, 0, 0, 0',
	X =	1840.921243	mm,	Y =	692.467965	mm,	Z =	806.136715	mm,
	W =	-120.782189	deg,	P =	-27.164001	deg,	R =	64.872909	deg
};
P[342]{
   GP1:
	UF : 0, UT : 1,		CONFIG : 'N U T, 0, 0, 0',
	X =	1856.015282	mm,	Y =	704.059203	mm,	Z =	800.881142	mm,
	W =	-122.075747	deg,	P =	-29.007907	deg,	R =	62.777602	deg
};
P[343]{
   GP1:
	UF : 0, UT : 1,		CONFIG : 'N U T, 0, 0, 0',
	X =	1871.750814	mm,	Y =	715.115572	mm,	Z =	796.323652	mm,
	W =	-123.796665	deg,	P =	-30.507452	deg,	R =	61.315682	deg
};
P[344]{
   GP1:
	UF : 0, UT : 1,		CONFIG : 'N U T, 0, 0, 0',
	X =	1888.125751	mm,	Y =	725.476187	mm,	Z =	792.635049	mm,
	W =	-126.804942	deg,	P =	-31.855386	deg,	R =	60.361948	deg
};
P[345]{
   GP1:
	UF : 0, UT : 1,		CONFIG : 'N U T, 0, 0, 0',
	X =	1905.132874	mm,	Y =	735.017482	mm,	Z =	789.764084	mm,
	W =	-129.228703	deg,	P =	-33.603873	deg,	R =	58.874018	deg
};
P[346]{
   GP1:
	UF : 0, UT : 1,		CONFIG : 'N U T, 0, 0, 0',
	X =	1922.727900	mm,	Y =	743.630220	mm,	Z =	787.812167	mm,
	W =	-131.377426	deg,	P =	-35.758333	deg,	R =	56.987025	deg
};
P[347]{
   GP1:
	UF : 0, UT : 1,		CONFIG : 'N U T, 0, 0, 0',
	X =	1940.860892	mm,	Y =	751.114036	mm,	Z =	787.032374	mm,
	W =	-134.605363	deg,	P =	-38.026981	deg,	R =	55.274931	deg
};
P[348]{
   GP1:
	UF : 0, UT : 1,		CONFIG : 'N U T, 0, 0, 0',
	X =	1959.442298	mm,	Y =	757.520864	mm,	Z =	787.314964	mm,
	W =	-137.913682	deg,	P =	-39.989483	deg,	R =	53.936419	deg
};
P[349]{
   GP1:
	UF : 0, UT : 1,		CONFIG : 'N U T, 0, 0, 0',
	X =	1978.306656	mm,	Y =	762.392975	mm,	Z =	788.979287	mm,
	W =	-142.012013	deg,	P =	-42.727639	deg,	R =	52.071295	deg
};
P[350]{
   GP1:
	UF : 0, UT : 1,		CONFIG : 'N U T, 0, 0, 0',
	X =	1997.374331	mm,	Y =	765.997682	mm,	Z =	791.834339	mm,
	W =	-146.387911	deg,	P =	-44.518675	deg,	R =	51.065699	deg
};
P[351]{
   GP1:
	UF : 0, UT : 1,		CONFIG : 'N U T, 0, 0, 0',
	X =	2016.430692	mm,	Y =	768.138965	mm,	Z =	795.846559	mm,
	W =	-150.125660	deg,	P =	-46.971978	deg,	R =	49.488091	deg
};
P[352]{
   GP1:
	UF : 0, UT : 1,		CONFIG : 'N U T, 0, 0, 0',
	X =	2035.277167	mm,	Y =	768.688191	mm,	Z =	801.071273	mm,
	W =	-153.367723	deg,	P =	-50.154894	deg,	R =	47.435468	deg
};
P[353]{
   GP1:
	UF : 0, UT : 1,		CONFIG : 'N U T, 0, 0, 0',
	X =	2053.836125	mm,	Y =	767.834989	mm,	Z =	807.342792	mm,
	W =	-155.775004	deg,	P =	-53.323700	deg,	R =	45.471900	deg
};
P[354]{
   GP1:
	UF : 0, UT : 1,		CONFIG : 'N U T, 0, 0, 0',
	X =	2071.840378	mm,	Y =	765.578300	mm,	Z =	814.739740	mm,
	W =	-159.603207	deg,	P =	-55.840080	deg,	R =	44.116673	deg
};
P[355]{
   GP1:
	UF : 0, UT : 1,		CONFIG : 'N U T, 0, 0, 0',
	X =	2089.347864	mm,	Y =	762.131211	mm,	Z =	822.993325	mm,
	W =	-163.023099	deg,	P =	-57.748119	deg,	R =	43.130372	deg
};
P[356]{
   GP1:
	UF : 0, UT : 1,		CONFIG : 'N U T, 0, 0, 0',
	X =	2106.271174	mm,	Y =	757.612757	mm,	Z =	831.978159	mm,
	W =	-166.295980	deg,	P =	-59.371866	deg,	R =	42.285031	deg
};
P[357]{
   GP1:
	UF : 0, UT : 1,		CONFIG : 'N U T, 0, 0, 0',
	X =	2122.415640	mm,	Y =	751.934511	mm,	Z =	841.654424	mm,
	W =	-169.255277	deg,	P =	-61.632766	deg,	R =	41.139979	deg
};
P[358]{
   GP1:
	UF : 0, UT : 1,		CONFIG : 'N U T, 0, 0, 0',
	X =	2138.022459	mm,	Y =	745.402968	mm,	Z =	851.843880	mm,
	W =	-171.195776	deg,	P =	-63.481355	deg,	R =	40.271553	deg
};
P[359]{
   GP1:
	UF : 0, UT : 1,		CONFIG : 'N U T, 0, 0, 0',
	X =	2152.835960	mm,	Y =	738.008479	mm,	Z =	862.552151	mm,
	W =	-173.683762	deg,	P =	-65.342682	deg,	R =	39.422502	deg
};
P[360]{
   GP1:
	UF : 0, UT : 1,		CONFIG : 'N U T, 0, 0, 0',
	X =	2167.116434	mm,	Y =	729.933303	mm,	Z =	873.621592	mm,
	W =	-175.221540	deg,	P =	-66.999933	deg,	R =	38.768972	deg
};
P[361]{
   GP1:
	UF : 0, UT : 1,		CONFIG : 'N U T, 0, 0, 0',
	X =	2180.690172	mm,	Y =	721.208560	mm,	Z =	885.049775	mm,
	W =	-177.158924	deg,	P =	-68.614910	deg,	R =	38.160644	deg
};
P[362]{
   GP1:
	UF : 0, UT : 1,		CONFIG : 'N U T, 0, 0, 0',
	X =	2193.260809	mm,	Y =	712.163140	mm,	Z =	896.466158	mm,
	W =	-179.111873	deg,	P =	-69.886868	deg,	R =	37.675763	deg
};
P[363]{
   GP1:
	UF : 0, UT : 1,		CONFIG : 'N U T, 0, 0, 0',
	X =	2199.935358	mm,	Y =	707.089929	mm,	Z =	902.721144	mm,
	W =	-179.818111	deg,	P =	-70.730950	deg,	R =	37.457435	deg
};
P[364]{
   GP1:
	UF : 0, UT : 1,		CONFIG : 'N U T, 0, 0, 0',
	X =	2197.209913	mm,	Y =	703.953533	mm,	Z =	891.166008	mm,
	W =	128.752361	deg,	P =	-57.696555	deg,	R =	93.373834	deg
};
P[365]{
   GP1:
	UF : 0, UT : 1,		CONFIG : 'N U T, 0, 0, 0',
	X =	2190.737141	mm,	Y =	708.852230	mm,	Z =	885.111108	mm,
	W =	128.752361	deg,	P =	-57.696555	deg,	R =	93.373834	deg
};
P[366]{
   GP1:
	UF : 0, UT : 1,		CONFIG : 'N U T, 0, 0, 0',
	X =	2177.749475	mm,	Y =	717.925282	mm,	Z =	873.567392	mm,
	W =	130.666511	deg,	P =	-57.546962	deg,	R =	93.332442	deg
};
P[367]{
   GP1:
	UF : 0, UT : 1,		CONFIG : 'N U T, 0, 0, 0',
	X =	2163.994788	mm,	Y =	726.375755	mm,	Z =	862.276104	mm,
	W =	133.491709	deg,	P =	-57.489112	deg,	R =	93.582151	deg
};
P[368]{
   GP1:
	UF : 0, UT : 1,		CONFIG : 'N U T, 0, 0, 0',
	X =	2149.632716	mm,	Y =	734.312169	mm,	Z =	851.325627	mm,
	W =	136.648247	deg,	P =	-56.855724	deg,	R =	92.682400	deg
};
P[369]{
   GP1:
	UF : 0, UT : 1,		CONFIG : 'N U T, 0, 0, 0',
	X =	2134.568011	mm,	Y =	741.370268	mm,	Z =	840.854596	mm,
	W =	140.522648	deg,	P =	-56.364901	deg,	R =	92.238921	deg
};
P[370]{
   GP1:
	UF : 0, UT : 1,		CONFIG : 'N U T, 0, 0, 0',
	X =	2118.886997	mm,	Y =	747.703505	mm,	Z =	830.756154	mm,
	W =	143.377125	deg,	P =	-56.413917	deg,	R =	92.514991	deg
};
P[371]{
   GP1:
	UF : 0, UT : 1,		CONFIG : 'N U T, 0, 0, 0',
	X =	2102.490128	mm,	Y =	752.980029	mm,	Z =	821.405026	mm,
	W =	148.225953	deg,	P =	-55.579306	deg,	R =	91.712723	deg
};
P[372]{
   GP1:
	UF : 0, UT : 1,		CONFIG : 'N U T, 0, 0, 0',
	X =	2085.496970	mm,	Y =	757.255732	mm,	Z =	812.516416	mm,
	W =	151.285936	deg,	P =	-56.676268	deg,	R =	92.888010	deg
};
P[373]{
   GP1:
	UF : 0, UT : 1,		CONFIG : 'N U T, 0, 0, 0',
	X =	2067.892796	mm,	Y =	760.549872	mm,	Z =	804.542376	mm,
	W =	156.415094	deg,	P =	-55.159220	deg,	R =	91.486753	deg
};
P[374]{
   GP1:
	UF : 0, UT : 1,		CONFIG : 'N U T, 0, 0, 0',
	X =	2049.779977	mm,	Y =	762.234700	mm,	Z =	797.486863	mm,
	W =	162.047761	deg,	P =	-56.052025	deg,	R =	91.859874	deg
};
P[375]{
   GP1:
	UF : 0, UT : 1,		CONFIG : 'N U T, 0, 0, 0',
	X =	2031.169595	mm,	Y =	762.760514	mm,	Z =	791.475884	mm,
	W =	167.401168	deg,	P =	-54.942517	deg,	R =	90.976356	deg
};
P[376]{
   GP1:
	UF : 0, UT : 1,		CONFIG : 'N U T, 0, 0, 0',
	X =	2012.301519	mm,	Y =	761.873025	mm,	Z =	786.481633	mm,
	W =	173.028839	deg,	P =	-54.668352	deg,	R =	90.472479	deg
};
P[377]{
   GP1:
	UF : 0, UT : 1,		CONFIG : 'N U T, 0, 0, 0',
	X =	1993.318566	mm,	Y =	759.460010	mm,	Z =	782.779126	mm,
	W =	179.370145	deg,	P =	-53.745834	deg,	R =	89.790338	deg
};
P[378]{
   GP1:
	UF : 0, UT : 1,		CONFIG : 'N U T, 0, 0, 0',
	X =	1974.331337	mm,	Y =	755.664654	mm,	Z =	780.143264	mm,
	W =	-174.786800	deg,	P =	-53.915056	deg,	R =	89.141397	deg
};
P[379]{
   GP1:
	UF : 0, UT : 1,		CONFIG : 'N U T, 0, 0, 0',
	X =	1955.650504	mm,	Y =	750.309799	mm,	Z =	778.855194	mm,
	W =	-167.442264	deg,	P =	-54.345338	deg,	R =	87.946564	deg
};
P[380]{
   GP1:
	UF : 0, UT : 1,		CONFIG : 'N U T, 0, 0, 0',
	X =	1937.232736	mm,	Y =	743.760442	mm,	Z =	778.821861	mm,
	W =	-162.039165	deg,	P =	-53.179595	deg,	R =	87.406548	deg
};
P[381]{
   GP1:
	UF : 0, UT : 1,		CONFIG : 'N U T, 0, 0, 0',
	X =	1919.293125	mm,	Y =	736.027359	mm,	Z =	779.845707	mm,
	W =	-156.385106	deg,	P =	-52.818781	deg,	R =	86.508453	deg
};
